    CONST robtarget rA_t278 := [[1931.75,1878.01,2213.21],[0.628788,0.0950822,0.552556,0.538765],[0,-2,-3,0],[9E+09,9E+09,9E+09,9E+09,9E+09,9E+09]];
    CONST robtarget rB_t278 := [[2895.21,136.965,1465.51],[0.672566,-0.676493,0.218304,-0.205806],[0,-3,2,0],[9E+09,9E+09,9E+09,9E+09,9E+09,9E+09]];
    CONST robtarget rB_t278_c1 := [[2895.21,136.965,1465.51],[0.672566,-0.676493,0.218304,-0.205806],[0,-4,-4,0],[9E+09,9E+09,9E+09,9E+09,9E+09,9E+09]];
    CONST robtarget rB_t278_c2 := [[2895.21,136.965,1465.51],[0.672566,-0.676493,0.218304,-0.205806],[0,0,-4,0],[9E+09,9E+09,9E+09,9E+09,9E+09,9E+09]];
    CONST jointtarget jA_t278 := [[44.9993,50.903,-73.3149,-90.0007,13.1401,-225.001],[9E+09,9E+09,9E+09,9E+09,9E+09,9E+09]];
    CONST jointtarget jB_t278 := [[0.000114317,56.0192,-54.9577,-270,55.0963,180],[9E+09,9E+09,9E+09,9E+09,9E+09,9E+09]];
    CONST jointtarget jBseed_t278 := [[0.000114414,56.0192,-54.9577,-270,55.0963,180],[9E+09,9E+09,9E+09,9E+09,9E+09,9E+09]];

    CONST robtarget rA_t279 := [[2895.21,136.965,1465.51],[0.672566,-0.676493,0.218304,-0.205806],[0,-3,2,0],[9E+09,9E+09,9E+09,9E+09,9E+09,9E+09]];
    CONST robtarget rB_t279 := [[1861.16,1900.88,2134.07],[0.550211,-0.0664014,0.550191,0.624619],[0,1,-2,0],[9E+09,9E+09,9E+09,9E+09,9E+09,9E+09]];
    CONST robtarget rB_t279_c4 := [[1861.16,1900.88,2134.07],[0.550211,-0.0664014,0.550191,0.624619],[0,-4,0,0],[9E+09,9E+09,9E+09,9E+09,9E+09,9E+09]];
    CONST robtarget rB_t279_c7 := [[1861.16,1900.88,2134.07],[0.550211,-0.0664014,0.550191,0.624619],[0,-4,4,0],[9E+09,9E+09,9E+09,9E+09,9E+09,9E+09]];
    CONST jointtarget jA_t279 := [[0.000114317,56.0192,-54.9577,-270,55.0963,180],[9E+09,9E+09,9E+09,9E+09,9E+09,9E+09]];
    CONST jointtarget jB_t279 := [[44.9999,40.5316,-53.7437,135,13.7626,-90.0002],[9E+09,9E+09,9E+09,9E+09,9E+09,9E+09]];
    CONST jointtarget jBseed_t279 := [[44.9999,40.5316,-53.7437,135,13.7626,-90.0001],[9E+09,9E+09,9E+09,9E+09,9E+09,9E+09]];

    CONST robtarget rA_t280 := [[1861.16,1900.88,2134.07],[0.550211,-0.0664014,0.550191,0.624619],[0,1,-2,0],[9E+09,9E+09,9E+09,9E+09,9E+09,9E+09]];
    CONST robtarget rB_t280 := [[89.7124,1202.36,2995.3],[0.131073,0.264977,0.137726,0.945325],[0,-2,2,0],[9E+09,9E+09,9E+09,9E+09,9E+09,9E+09]];
    CONST robtarget rB_t280_c1 := [[89.7124,1202.36,2995.3],[0.131073,0.264977,0.137726,0.945325],[0,-4,-4,0],[9E+09,9E+09,9E+09,9E+09,9E+09,9E+09]];
    CONST robtarget rB_t280_c2 := [[89.7124,1202.36,2995.3],[0.131073,0.264977,0.137726,0.945325],[0,0,-4,0],[9E+09,9E+09,9E+09,9E+09,9E+09,9E+09]];
    CONST jointtarget jA_t280 := [[44.9999,40.5316,-53.7437,135,13.7626,-90.0002],[9E+09,9E+09,9E+09,9E+09,9E+09,9E+09]];
    CONST jointtarget jB_t280 := [[89.999,-13.3177,-24.0516,-135.001,49.4253,224.999],[9E+09,9E+09,9E+09,9E+09,9E+09,9E+09]];
    CONST jointtarget jBseed_t280 := [[89.999,-13.3177,-24.0516,-135.001,49.4253,224.999],[9E+09,9E+09,9E+09,9E+09,9E+09,9E+09]];

    CONST robtarget rA_t281 := [[89.7124,1202.36,2995.3],[0.131073,0.264977,0.137726,0.945325],[0,-2,2,0],[9E+09,9E+09,9E+09,9E+09,9E+09,9E+09]];
    CONST robtarget rB_t281 := [[8.43678,485.853,3488.8],[0.00349083,0.0250045,0.137295,0.990208],[0,2,1,0],[9E+09,9E+09,9E+09,9E+09,9E+09,9E+09]];
    CONST robtarget rB_t281_c5 := [[8.43678,485.853,3488.8],[0.00349083,0.0250045,0.137295,0.990208],[0,0,0,0],[9E+09,9E+09,9E+09,9E+09,9E+09,9E+09]];
    CONST jointtarget jA_t281 := [[89.999,-13.3177,-24.0516,-135.001,49.4253,224.999],[9E+09,9E+09,9E+09,9E+09,9E+09,9E+09]];
    CONST jointtarget jB_t281 := [[89.9991,-5.53912,-68.673,269.999,2.89315,179.999],[9E+09,9E+09,9E+09,9E+09,9E+09,9E+09]];
    CONST jointtarget jBseed_t281 := [[89.9991,-5.53911,-68.6731,269.999,2.89315,179.999],[9E+09,9E+09,9E+09,9E+09,9E+09,9E+09]];

    CONST robtarget rA_t283 := [[-1405.69,-1439.34,2692.16],[0.0384433,0.29226,0.377677,-0.877762],[-2,1,2,0],[9E+09,9E+09,9E+09,9E+09,9E+09,9E+09]];
    CONST robtarget rB_t283 := [[812.974,-812.948,3221.93],[0.912154,0.146672,0.0607486,0.377853],[-1,2,-1,0],[9E+09,9E+09,9E+09,9E+09,9E+09,9E+09]];
    CONST robtarget rB_t283_c5 := [[812.974,-812.948,3221.93],[0.912154,0.146672,0.0607486,0.377853],[0,0,0,0],[9E+09,9E+09,9E+09,9E+09,9E+09,9E+09]];
    CONST robtarget rB_t283_c8 := [[812.974,-812.948,3221.93],[0.912154,0.146672,0.0607486,0.377853],[0,0,4,0],[9E+09,9E+09,9E+09,9E+09,9E+09,9E+09]];
    CONST jointtarget jA_t283 := [[-135,12.1897,-37.2472,135,11.6221,180],[9E+09,9E+09,9E+09,9E+09,9E+09,9E+09]];
    CONST jointtarget jB_t283 := [[-44.999,-5.94196,-41.7701,180.001,24.0187,-89.999],[9E+09,9E+09,9E+09,9E+09,9E+09,9E+09]];
    CONST jointtarget jBseed_t283 := [[-44.999,-5.94196,-41.7701,180.001,24.0187,-89.999],[9E+09,9E+09,9E+09,9E+09,9E+09,9E+09]];

    CONST robtarget rA_t284 := [[812.974,-812.948,3221.93],[0.912154,0.146672,0.0607486,0.377853],[-1,2,-1,0],[9E+09,9E+09,9E+09,9E+09,9E+09,9E+09]];
    CONST robtarget rB_t284 := [[1979.94,1852.8,2089.61],[0.764614,0.235393,0.316893,0.509445],[0,-2,-2,0],[9E+09,9E+09,9E+09,9E+09,9E+09,9E+09]];
    CONST robtarget rB_t284_c2 := [[1979.94,1852.8,2089.61],[0.764614,0.235393,0.316893,0.509445],[0,0,-4,0],[9E+09,9E+09,9E+09,9E+09,9E+09,9E+09]];
    CONST robtarget rB_t284_c3 := [[1979.94,1852.8,2089.61],[0.764614,0.235393,0.316893,0.509445],[0,4,-4,0],[9E+09,9E+09,9E+09,9E+09,9E+09,9E+09]];
    CONST jointtarget jA_t284 := [[-44.999,-5.94196,-41.7701,180.001,24.0187,-89.999],[9E+09,9E+09,9E+09,9E+09,9E+09,9E+09]];
    CONST jointtarget jB_t284 := [[45.0006,50.687,-65.7411,-134.999,49.5993,-179.999],[9E+09,9E+09,9E+09,9E+09,9E+09,9E+09]];
    CONST jointtarget jBseed_t284 := [[45.0006,50.687,-65.7411,-134.999,49.5993,-179.999],[9E+09,9E+09,9E+09,9E+09,9E+09,9E+09]];

    CONST robtarget rA_t286 := [[-1258.34,-1258.33,725.886],[0.308285,0.870927,-0.360749,-0.127697],[-2,-1,-4,0],[9E+09,9E+09,9E+09,9E+09,9E+09,9E+09]];
    CONST robtarget rB_t286 := [[767.091,-675.421,2450.3],[0.568653,0.350797,0.169976,0.72435],[-1,-3,-4,0],[9E+09,9E+09,9E+09,9E+09,9E+09,9E+09]];
    CONST robtarget rB_t286_c2 := [[767.091,-675.421,2450.3],[0.568653,0.350797,0.169976,0.72435],[0,0,-4,0],[9E+09,9E+09,9E+09,9E+09,9E+09,9E+09]];
    CONST jointtarget jA_t286 := [[-135,5.1912,38.7445,-0.000157696,7.07907,-270],[9E+09,9E+09,9E+09,9E+09,9E+09,9E+09]];
    CONST jointtarget jB_t286 := [[-44.9991,-40.7514,16.6024,-224.999,33.2841,-359.999],[9E+09,9E+09,9E+09,9E+09,9E+09,9E+09]];
    CONST jointtarget jBseed_t286 := [[-44.9991,-40.7514,16.6024,-224.999,33.2841,-359.999],[9E+09,9E+09,9E+09,9E+09,9E+09,9E+09]];

    CONST robtarget rA_t288 := [[-39.7659,1340.08,1419.52],[0.53573,-0.738869,-0.390158,-0.121829],[1,0,2,0],[9E+09,9E+09,9E+09,9E+09,9E+09,9E+09]];
    CONST robtarget rB_t288 := [[12.6582,1912.94,1121.44],[0.311805,-0.635779,-0.608576,-0.358048],[0,-1,2,0],[9E+09,9E+09,9E+09,9E+09,9E+09,9E+09]];
    CONST robtarget rB_t288_c5 := [[12.6582,1912.94,1121.44],[0.311805,-0.635779,-0.608576,-0.358048],[0,0,0,0],[9E+09,9E+09,9E+09,9E+09,9E+09,9E+09]];
    CONST jointtarget jA_t288 := [[90.0009,-37.8252,47.7227,45.0009,19.668,180.001],[9E+09,9E+09,9E+09,9E+09,9E+09,9E+09]];
    CONST jointtarget jB_t288 := [[89.9998,0.210577,28.8498,-45.0002,6.1507,225],[9E+09,9E+09,9E+09,9E+09,9E+09,9E+09]];
    CONST jointtarget jBseed_t288 := [[89.9998,0.210579,28.8498,-45.0002,6.1507,225],[9E+09,9E+09,9E+09,9E+09,9E+09,9E+09]];

    CONST robtarget rA_t290 := [[1406.56,-1559.53,2818.3],[0.150617,0.0701145,-0.509223,0.844447],[-1,3,-1,0],[9E+09,9E+09,9E+09,9E+09,9E+09,9E+09]];
    CONST robtarget rB_t290 := [[1821.8,-1916.48,1910.44],[0.145501,-0.116653,0.673226,-0.715534],[-1,2,-5,0],[9E+09,9E+09,9E+09,9E+09,9E+09,9E+09]];
    CONST robtarget rB_t290_c5 := [[1821.8,-1916.48,1910.44],[0.145501,-0.116653,0.673226,-0.715534],[0,0,0,0],[9E+09,9E+09,9E+09,9E+09,9E+09,9E+09]];
    CONST robtarget rB_t290_c6 := [[1821.8,-1916.48,1910.44],[0.145501,-0.116653,0.673226,-0.715534],[0,4,0,0],[9E+09,9E+09,9E+09,9E+09,9E+09,9E+09]];
    CONST jointtarget jA_t290 := [[-44.9996,31.5372,-69.78,270,40.376,-44.9996],[9E+09,9E+09,9E+09,9E+09,9E+09,9E+09]];
    CONST jointtarget jB_t290 := [[-45.0008,34.9614,-39.1119,269.999,23.6195,-360.001],[9E+09,9E+09,9E+09,9E+09,9E+09,9E+09]];
    CONST jointtarget jBseed_t290 := [[-45.0008,34.9614,-39.1119,269.999,23.6195,-360.001],[9E+09,9E+09,9E+09,9E+09,9E+09,9E+09]];

    CONST robtarget rA_t291 := [[1821.8,-1916.48,1910.44],[0.145501,-0.116653,0.673226,-0.715534],[-1,2,-5,0],[9E+09,9E+09,9E+09,9E+09,9E+09,9E+09]];
    CONST robtarget rB_t291 := [[50.5098,-2702.01,2116.99],[0.762943,0.487354,-0.0695059,0.419015],[-1,1,-4,0],[9E+09,9E+09,9E+09,9E+09,9E+09,9E+09]];
    CONST robtarget rB_t291_c5 := [[50.5098,-2702.01,2116.99],[0.762943,0.487354,-0.0695059,0.419015],[0,0,0,0],[9E+09,9E+09,9E+09,9E+09,9E+09,9E+09]];
    CONST jointtarget jA_t291 := [[-45.0008,34.9614,-39.1119,269.999,23.6195,-360.001],[9E+09,9E+09,9E+09,9E+09,9E+09,9E+09]];
    CONST jointtarget jB_t291 := [[-89.9996,45.3841,-59.6154,135,25.3151,-360],[9E+09,9E+09,9E+09,9E+09,9E+09,9E+09]];
    CONST jointtarget jBseed_t291 := [[-89.9996,45.3841,-59.6155,135,25.3151,-360],[9E+09,9E+09,9E+09,9E+09,9E+09,9E+09]];

    CONST robtarget rA_t293 := [[0.000160017,-2033.22,1759.97],[8.87382E-8,3.03818E-8,0.817508,-0.575917],[-1,0,3,0],[9E+09,9E+09,9E+09,9E+09,9E+09,9E+09]];
    CONST robtarget rB_t293 := [[-705.743,-705.745,3293.67],[2.528E-6,-0.101964,-0.101965,-0.989549],[-2,2,-3,0],[9E+09,9E+09,9E+09,9E+09,9E+09,9E+09]];
    CONST robtarget rB_t293_c5 := [[-705.743,-705.745,3293.67],[2.528E-6,-0.101964,-0.101965,-0.989549],[0,0,0,0],[9E+09,9E+09,9E+09,9E+09,9E+09,9E+09]];
    CONST jointtarget jA_t293 := [[-90,-0.214244,6.61641,9.73535E-6,13.2701,270],[9E+09,9E+09,9E+09,9E+09,9E+09,9E+09]];
    CONST jointtarget jB_t293 := [[-135,-3.3015,-48.9074,180,54.373,-225],[9E+09,9E+09,9E+09,9E+09,9E+09,9E+09]];
    CONST jointtarget jBseed_t293 := [[-135,-3.30149,-48.9074,180,54.373,-225],[9E+09,9E+09,9E+09,9E+09,9E+09,9E+09]];

    CONST robtarget rA_t294 := [[-705.743,-705.745,3293.67],[2.528E-6,-0.101964,-0.101965,-0.989549],[-2,2,-3,0],[9E+09,9E+09,9E+09,9E+09,9E+09,9E+09]];
    CONST robtarget rB_t294 := [[-1094.14,-971.928,9.47825],[0.208069,-0.895798,-0.340492,0.195752],[-2,3,1,0],[9E+09,9E+09,9E+09,9E+09,9E+09,9E+09]];
    CONST robtarget rB_t294_c3 := [[-1094.14,-971.928,9.47825],[0.208069,-0.895798,-0.340492,0.195752],[0,4,-4,0],[9E+09,9E+09,9E+09,9E+09,9E+09,9E+09]];
    CONST jointtarget jA_t294 := [[-135,-3.3015,-48.9074,180,54.373,-225],[9E+09,9E+09,9E+09,9E+09,9E+09,9E+09]];
    CONST jointtarget jB_t294 := [[-135,31.9108,46.0247,270,31.1655,90.0004],[9E+09,9E+09,9E+09,9E+09,9E+09,9E+09]];
    CONST jointtarget jBseed_t294 := [[-135,31.9108,46.0247,270,31.1655,90.0004],[9E+09,9E+09,9E+09,9E+09,9E+09,9E+09]];

    CONST robtarget rA_t295 := [[-1094.14,-971.928,9.47825],[0.208069,-0.895798,-0.340492,0.195752],[-2,3,1,0],[9E+09,9E+09,9E+09,9E+09,9E+09,9E+09]];
    CONST robtarget rB_t295 := [[-0.0128204,-2555.07,2364.03],[0.379873,0.046241,0.111641,-0.917112],[-2,-3,1,0],[9E+09,9E+09,9E+09,9E+09,9E+09,9E+09]];
    CONST robtarget rB_t295_c5 := [[-0.0128204,-2555.07,2364.03],[0.379873,0.046241,0.111641,-0.917112],[0,0,0,0],[9E+09,9E+09,9E+09,9E+09,9E+09,9E+09]];
    CONST jointtarget jA_t295 := [[-135,31.9108,46.0247,270,31.1655,90.0004],[9E+09,9E+09,9E+09,9E+09,9E+09,9E+09]];
    CONST jointtarget jB_t295 := [[-90.0003,51.5513,-76.5603,-180,51.1099,135],[9E+09,9E+09,9E+09,9E+09,9E+09,9E+09]];
    CONST jointtarget jBseed_t295 := [[-90.0003,51.5513,-76.5603,-180,51.11,135],[9E+09,9E+09,9E+09,9E+09,9E+09,9E+09]];

    CONST robtarget rA_t296 := [[-0.0128204,-2555.07,2364.03],[0.379873,0.046241,0.111641,-0.917112],[-2,-3,1,0],[9E+09,9E+09,9E+09,9E+09,9E+09,9E+09]];
    CONST robtarget rB_t296 := [[-133.882,-1999.9,2604.31],[0.245559,-0.3752,-0.489462,0.747899],[-2,-2,-1,0],[9E+09,9E+09,9E+09,9E+09,9E+09,9E+09]];
    CONST robtarget rB_t296_c5 := [[-133.882,-1999.9,2604.31],[0.245559,-0.3752,-0.489462,0.747899],[0,0,0,0],[9E+09,9E+09,9E+09,9E+09,9E+09,9E+09]];
    CONST jointtarget jA_t296 := [[-90.0003,51.5513,-76.5603,-180,51.1099,135],[9E+09,9E+09,9E+09,9E+09,9E+09,9E+09]];
    CONST jointtarget jB_t296 := [[-90.0004,12.9148,-36.5093,-90.0004,53.2835,-0.000410538],[9E+09,9E+09,9E+09,9E+09,9E+09,9E+09]];
    CONST jointtarget jBseed_t296 := [[-90.0004,12.9148,-36.5093,-90.0004,53.2835,-0.000407697],[9E+09,9E+09,9E+09,9E+09,9E+09,9E+09]];

    CONST robtarget rA_t297 := [[-133.882,-1999.9,2604.31],[0.245559,-0.3752,-0.489462,0.747899],[-2,-2,-1,0],[9E+09,9E+09,9E+09,9E+09,9E+09,9E+09]];
    CONST robtarget rB_t297 := [[1996.66,-62.2443,1865.38],[0.57107,0.599825,0.416979,0.374455],[0,3,-2,0],[9E+09,9E+09,9E+09,9E+09,9E+09,9E+09]];
    CONST robtarget rB_t297_c2 := [[1996.66,-62.2443,1865.38],[0.57107,0.599825,0.416979,0.374455],[0,0,-4,0],[9E+09,9E+09,9E+09,9E+09,9E+09,9E+09]];
    CONST robtarget rB_t297_c5 := [[1996.66,-62.2443,1865.38],[0.57107,0.599825,0.416979,0.374455],[0,0,0,0],[9E+09,9E+09,9E+09,9E+09,9E+09,9E+09]];
    CONST jointtarget jA_t297 := [[-90.0004,12.9148,-36.5093,-90.0004,53.2835,-0.000410538],[9E+09,9E+09,9E+09,9E+09,9E+09,9E+09]];
    CONST jointtarget jB_t297 := [[0.000436422,-1.83294,5.99353,270,21.8891,-180],[9E+09,9E+09,9E+09,9E+09,9E+09,9E+09]];
    CONST jointtarget jBseed_t297 := [[0.000436628,-1.83294,5.99353,270,21.8891,-180],[9E+09,9E+09,9E+09,9E+09,9E+09,9E+09]];

    CONST robtarget rA_t298 := [[1996.66,-62.2443,1865.38],[0.57107,0.599825,0.416979,0.374455],[0,3,-2,0],[9E+09,9E+09,9E+09,9E+09,9E+09,9E+09]];
    CONST robtarget rB_t298 := [[-0.0358595,2407.99,2512.57],[0.694216,-0.134324,0.134333,0.694245],[1,2,2,0],[9E+09,9E+09,9E+09,9E+09,9E+09,9E+09]];
    CONST robtarget rB_t298_c2 := [[-0.0358595,2407.99,2512.57],[0.694216,-0.134324,0.134333,0.694245],[0,0,-4,0],[9E+09,9E+09,9E+09,9E+09,9E+09,9E+09]];
    CONST jointtarget jA_t298 := [[0.000436422,-1.83294,5.99353,270,21.8891,-180],[9E+09,9E+09,9E+09,9E+09,9E+09,9E+09]];
    CONST jointtarget jB_t298 := [[90.0009,37.9388,-61.6031,180.001,44.4337,180.001],[9E+09,9E+09,9E+09,9E+09,9E+09,9E+09]];
    CONST jointtarget jBseed_t298 := [[90.0009,37.9388,-61.6031,180.001,44.4337,180.001],[9E+09,9E+09,9E+09,9E+09,9E+09,9E+09]];

    CONST robtarget rA_t299 := [[-0.0358595,2407.99,2512.57],[0.694216,-0.134324,0.134333,0.694245],[1,2,2,0],[9E+09,9E+09,9E+09,9E+09,9E+09,9E+09]];
    CONST robtarget rB_t299 := [[0.0269352,2024.98,2914.37],[0.65455,-0.267481,-0.267485,-0.654576],[0,-3,3,0],[9E+09,9E+09,9E+09,9E+09,9E+09,9E+09]];
    CONST robtarget rB_t299_c5 := [[0.0269352,2024.98,2914.37],[0.65455,-0.267481,-0.267485,-0.654576],[0,0,0,0],[9E+09,9E+09,9E+09,9E+09,9E+09,9E+09]];
    CONST robtarget rB_t299_c8 := [[0.0269352,2024.98,2914.37],[0.65455,-0.267481,-0.267485,-0.654576],[0,0,4,0],[9E+09,9E+09,9E+09,9E+09,9E+09,9E+09]];
    CONST jointtarget jA_t299 := [[90.0009,37.9388,-61.6031,180.001,44.4337,180.001],[9E+09,9E+09,9E+09,9E+09,9E+09,9E+09]];
    CONST jointtarget jB_t299 := [[89.9992,27.0766,-66.003,-180.001,6.61947,359.999],[9E+09,9E+09,9E+09,9E+09,9E+09,9E+09]];
    CONST jointtarget jBseed_t299 := [[89.9992,27.0766,-66.003,-180.001,6.61946,359.999],[9E+09,9E+09,9E+09,9E+09,9E+09,9E+09]];

    CONST robtarget rA_t301 := [[711.687,820.474,2264.17],[0.740004,-0.357438,-0.197934,-0.534279],[0,1,-4,0],[9E+09,9E+09,9E+09,9E+09,9E+09,9E+09]];
    CONST robtarget rB_t301 := [[-794.783,716.383,3401.08],[0.401784,0.232779,-0.132142,-0.875741],[1,-4,-1,0],[9E+09,9E+09,9E+09,9E+09,9E+09,9E+09]];
    CONST robtarget rB_t301_c5 := [[-794.783,716.383,3401.08],[0.401784,0.232779,-0.132142,-0.875741],[0,0,0,0],[9E+09,9E+09,9E+09,9E+09,9E+09,9E+09]];
    CONST jointtarget jA_t301 := [[44.9993,-42.165,24.799,134.999,40.6561,-270.001],[9E+09,9E+09,9E+09,9E+09,9E+09,9E+09]];
    CONST jointtarget jB_t301 := [[135,11.1533,-76.4135,-270,19.3896,-0.000262528],[9E+09,9E+09,9E+09,9E+09,9E+09,9E+09]];
    CONST jointtarget jBseed_t301 := [[135,11.1533,-76.4135,-270,19.3896,-0.000243019],[9E+09,9E+09,9E+09,9E+09,9E+09,9E+09]];

    CONST robtarget rA_t303 := [[-1207.94,-1217.23,2595.23],[0.584806,0.577737,0.0162937,-0.569172],[-2,0,3,0],[9E+09,9E+09,9E+09,9E+09,9E+09,9E+09]];
    CONST robtarget rB_t303 := [[-1933.3,-2020.07,1434.77],[0.640752,0.612752,-0.440334,0.141698],[-2,-3,0,0],[9E+09,9E+09,9E+09,9E+09,9E+09,9E+09]];
    CONST robtarget rB_t303_c5 := [[-1933.3,-2020.07,1434.77],[0.640752,0.612752,-0.440334,0.141698],[0,0,0,0],[9E+09,9E+09,9E+09,9E+09,9E+09,9E+09]];
    CONST jointtarget jA_t303 := [[-135,-6.5096,-15.1488,44.9998,3.19163,360],[9E+09,9E+09,9E+09,9E+09,9E+09,9E+09]];
    CONST jointtarget jB_t303 := [[-135,42.8608,-34.2836,-270,21.5467,45.0005],[9E+09,9E+09,9E+09,9E+09,9E+09,9E+09]];
    CONST jointtarget jBseed_t303 := [[-135,42.8608,-34.2836,-270,21.5467,45.0005],[9E+09,9E+09,9E+09,9E+09,9E+09,9E+09]];

    CONST robtarget rA_t306 := [[-0.00435252,-1330.24,-413.892],[0.081587,0.373884,0.902639,-0.196969],[-2,1,-3,0],[9E+09,9E+09,9E+09,9E+09,9E+09,9E+09]];
    CONST robtarget rB_t306 := [[1109.78,-1031.5,1346.08],[0.314617,0.796486,0.0990844,0.506762],[-1,0,0,0],[9E+09,9E+09,9E+09,9E+09,9E+09,9E+09]];
    CONST robtarget rB_t306_c2 := [[1109.78,-1031.5,1346.08],[0.314617,0.796486,0.0990844,0.506762],[0,0,-4,0],[9E+09,9E+09,9E+09,9E+09,9E+09,9E+09]];
    CONST robtarget rB_t306_c5 := [[1109.78,-1031.5,1346.08],[0.314617,0.796486,0.0990844,0.506762],[0,0,0,0],[9E+09,9E+09,9E+09,9E+09,9E+09,9E+09]];
    CONST jointtarget jA_t306 := [[-90.0002,55.88,40.99,180,31.4896,-225],[9E+09,9E+09,9E+09,9E+09,9E+09,9E+09]];
    CONST jointtarget jB_t306 := [[-45.0005,-25.9706,43.7712,89.9995,19.3622,44.9995],[9E+09,9E+09,9E+09,9E+09,9E+09,9E+09]];
    CONST jointtarget jBseed_t306 := [[-45.0005,-25.9706,43.7712,89.9995,19.3622,44.9995],[9E+09,9E+09,9E+09,9E+09,9E+09,9E+09]];

    CONST robtarget rA_t307 := [[1109.78,-1031.5,1346.08],[0.314617,0.796486,0.0990844,0.506762],[-1,0,0,0],[9E+09,9E+09,9E+09,9E+09,9E+09,9E+09]];
    CONST robtarget rB_t307 := [[1813.28,-1813.32,1534.44],[0.580903,0.575562,0.575569,-1.19777E-5],[-1,-1,0,0],[9E+09,9E+09,9E+09,9E+09,9E+09,9E+09]];
    CONST robtarget rB_t307_c5 := [[1813.28,-1813.32,1534.44],[0.580903,0.575562,0.575569,-1.19777E-5],[0,0,0,0],[9E+09,9E+09,9E+09,9E+09,9E+09,9E+09]];
    CONST jointtarget jA_t307 := [[-45.0005,-25.9706,43.7712,89.9995,19.3622,44.9995],[9E+09,9E+09,9E+09,9E+09,9E+09,9E+09]];
    CONST jointtarget jB_t307 := [[-45.0007,28.1057,-18.1997,-0.000729667,9.06583,44.9993],[9E+09,9E+09,9E+09,9E+09,9E+09,9E+09]];
    CONST jointtarget jBseed_t307 := [[-45.0007,28.1057,-18.1997,-0.000737297,9.06583,44.9993],[9E+09,9E+09,9E+09,9E+09,9E+09,9E+09]];

    CONST robtarget rA_t308 := [[1813.28,-1813.32,1534.44],[0.580903,0.575562,0.575569,-1.19777E-5],[-1,-1,0,0],[9E+09,9E+09,9E+09,9E+09,9E+09,9E+09]];
    CONST robtarget rB_t308 := [[2140.65,93.5238,2492.89],[0.519043,-0.360662,-0.121204,-0.765393],[0,-3,-3,0],[9E+09,9E+09,9E+09,9E+09,9E+09,9E+09]];
    CONST robtarget rB_t308_c4 := [[2140.65,93.5238,2492.89],[0.519043,-0.360662,-0.121204,-0.765393],[0,-4,0,0],[9E+09,9E+09,9E+09,9E+09,9E+09,9E+09]];
    CONST robtarget rB_t308_c5 := [[2140.65,93.5238,2492.89],[0.519043,-0.360662,-0.121204,-0.765393],[0,0,0,0],[9E+09,9E+09,9E+09,9E+09,9E+09,9E+09]];
    CONST jointtarget jA_t308 := [[-45.0007,28.1057,-18.1997,-0.000729667,9.06583,44.9993],[9E+09,9E+09,9E+09,9E+09,9E+09,9E+09]];
    CONST jointtarget jB_t308 := [[0.000401838,16.7455,-33.264,-225,52.3606,-270],[9E+09,9E+09,9E+09,9E+09,9E+09,9E+09]];
    CONST jointtarget jBseed_t308 := [[0.000401837,16.7455,-33.264,-225,52.3606,-270],[9E+09,9E+09,9E+09,9E+09,9E+09,9E+09]];

    CONST robtarget rA_t311 := [[-1668.51,-1668.47,341.824],[0.590053,0.294475,-0.710909,0.2444],[-2,-3,3,0],[9E+09,9E+09,9E+09,9E+09,9E+09,9E+09]];
    CONST robtarget rB_t311 := [[1659.54,-1659.53,736.873],[0.559459,7.7831E-7,0.611567,-0.559457],[-1,-2,-3,0],[9E+09,9E+09,9E+09,9E+09,9E+09,9E+09]];
    CONST robtarget rB_t311_c4 := [[1659.54,-1659.53,736.873],[0.559459,7.7831E-7,0.611567,-0.559457],[0,-4,0,0],[9E+09,9E+09,9E+09,9E+09,9E+09,9E+09]];
    CONST jointtarget jA_t311 := [[-135.001,43.7764,8.73104,-180.001,41.8922,359.999],[9E+09,9E+09,9E+09,9E+09,9E+09,9E+09]];
    CONST jointtarget jB_t311 := [[-44.9999,32.6286,10.7941,-180,58.0169,-225],[9E+09,9E+09,9E+09,9E+09,9E+09,9E+09]];
    CONST jointtarget jBseed_t311 := [[-44.9999,32.6286,10.7941,-180,58.0169,-225],[9E+09,9E+09,9E+09,9E+09,9E+09,9E+09]];

    CONST robtarget rA_t316 := [[31.8866,-661.423,2881.06],[0.650157,0.260758,0.387274,-0.599433],[-2,0,-1,0],[9E+09,9E+09,9E+09,9E+09,9E+09,9E+09]];
    CONST robtarget rB_t316 := [[67.0004,-1549.03,-423.181],[0.0272108,0.674661,0.686619,0.269531],[-1,0,-1,0],[9E+09,9E+09,9E+09,9E+09,9E+09,9E+09]];
    CONST robtarget rB_t316_c5 := [[67.0004,-1549.03,-423.181],[0.0272108,0.674661,0.686619,0.269531],[0,0,0,0],[9E+09,9E+09,9E+09,9E+09,9E+09,9E+09]];
    CONST jointtarget jA_t316 := [[-90.0005,-39.8358,-6.45618,44.9995,15.6688,-45.0005],[9E+09,9E+09,9E+09,9E+09,9E+09,9E+09]];
    CONST jointtarget jB_t316 := [[-89.9991,59.0698,26.3106,45.0009,34.5531,-44.9991],[9E+09,9E+09,9E+09,9E+09,9E+09,9E+09]];
    CONST jointtarget jBseed_t316 := [[-89.9991,59.0698,26.3106,45.0009,34.5531,-44.9991],[9E+09,9E+09,9E+09,9E+09,9E+09,9E+09]];

    CONST robtarget rA_t317 := [[67.0004,-1549.03,-423.181],[0.0272108,0.674661,0.686619,0.269531],[-1,0,-1,0],[9E+09,9E+09,9E+09,9E+09,9E+09,9E+09]];
    CONST robtarget rB_t317 := [[1093.81,-961.271,-433.788],[0.203083,0.00193774,0.955933,0.212005],[-1,-3,-2,0],[9E+09,9E+09,9E+09,9E+09,9E+09,9E+09]];
    CONST robtarget rB_t317_c5 := [[1093.81,-961.271,-433.788],[0.203083,0.00193774,0.955933,0.212005],[0,0,0,0],[9E+09,9E+09,9E+09,9E+09,9E+09,9E+09]];
    CONST robtarget rB_t317_c8 := [[1093.81,-961.271,-433.788],[0.203083,0.00193774,0.955933,0.212005],[0,0,4,0],[9E+09,9E+09,9E+09,9E+09,9E+09,9E+09]];
    CONST jointtarget jA_t317 := [[-89.9991,59.0698,26.3106,45.0009,34.5531,-44.9991],[9E+09,9E+09,9E+09,9E+09,9E+09,9E+09]];
    CONST jointtarget jB_t317 := [[-44.9999,58.5461,32.2102,-270,34.1374,-135],[9E+09,9E+09,9E+09,9E+09,9E+09,9E+09]];
    CONST jointtarget jBseed_t317 := [[-44.9999,58.5461,32.2102,-270,34.1374,-135],[9E+09,9E+09,9E+09,9E+09,9E+09,9E+09]];

    CONST robtarget rA_t319 := [[-247.85,152.002,3494.48],[0.3863,0.144348,0.205674,-0.887488],[1,-3,-1,0],[9E+09,9E+09,9E+09,9E+09,9E+09,9E+09]];
    CONST robtarget rB_t319 := [[1522.3,1582.86,1574.78],[0.437235,-0.846027,-0.0820903,-0.293813],[0,0,1,0],[9E+09,9E+09,9E+09,9E+09,9E+09,9E+09]];
    CONST robtarget rB_t319_c2 := [[1522.3,1582.86,1574.78],[0.437235,-0.846027,-0.0820903,-0.293813],[0,0,-4,0],[9E+09,9E+09,9E+09,9E+09,9E+09,9E+09]];
    CONST jointtarget jA_t319 := [[135.001,-2.30911,-78.3931,-224.999,35.0237,-44.9992],[9E+09,9E+09,9E+09,9E+09,9E+09,9E+09]];
    CONST jointtarget jB_t319 := [[44.9998,9.10246,2.92276,44.9998,21.2665,180],[9E+09,9E+09,9E+09,9E+09,9E+09,9E+09]];
    CONST jointtarget jBseed_t319 := [[44.9998,9.10246,2.92276,44.9998,21.2665,180],[9E+09,9E+09,9E+09,9E+09,9E+09,9E+09]];

    CONST robtarget rA_t320 := [[1522.3,1582.86,1574.78],[0.437235,-0.846027,-0.0820903,-0.293813],[0,0,1,0],[9E+09,9E+09,9E+09,9E+09,9E+09,9E+09]];
    CONST robtarget rB_t320 := [[29.1179,-2091.95,2261.12],[0.459763,0.544345,-0.448947,0.539215],[-1,0,1,0],[9E+09,9E+09,9E+09,9E+09,9E+09,9E+09]];
    CONST robtarget rB_t320_c5 := [[29.1179,-2091.95,2261.12],[0.459763,0.544345,-0.448947,0.539215],[0,0,0,0],[9E+09,9E+09,9E+09,9E+09,9E+09,9E+09]];
    CONST jointtarget jA_t320 := [[44.9998,9.10246,2.92276,44.9998,21.2665,180],[9E+09,9E+09,9E+09,9E+09,9E+09,9E+09]];
    CONST jointtarget jB_t320 := [[-89.9993,6.24591,-16.6842,45.0007,14.2625,135.001],[9E+09,9E+09,9E+09,9E+09,9E+09,9E+09]];
    CONST jointtarget jBseed_t320 := [[-89.9993,6.24592,-16.6842,45.0007,14.2625,135.001],[9E+09,9E+09,9E+09,9E+09,9E+09,9E+09]];

    CONST robtarget rA_t322 := [[-0.0284785,1965.77,2672.38],[1.9163E-5,-6.84607E-6,-0.149469,-0.988766],[1,2,3,0],[9E+09,9E+09,9E+09,9E+09,9E+09,9E+09]];
    CONST robtarget rB_t322 := [[42.8658,1982.85,2907.31],[0.887318,-0.257326,0.232757,0.303767],[1,-2,-3,0],[9E+09,9E+09,9E+09,9E+09,9E+09,9E+09]];
    CONST robtarget rB_t322_c6 := [[42.8658,1982.85,2907.31],[0.887318,-0.257326,0.232757,0.303767],[0,4,0,0],[9E+09,9E+09,9E+09,9E+09,9E+09,9E+09]];
    CONST jointtarget jA_t322 := [[90.0009,11.6331,-32.8236,180.001,51.6172,270.001],[9E+09,9E+09,9E+09,9E+09,9E+09,9E+09]];
    CONST jointtarget jB_t322 := [[90.0002,22.8797,-59.2465,-135,21.2885,-270],[9E+09,9E+09,9E+09,9E+09,9E+09,9E+09]];
    CONST jointtarget jBseed_t322 := [[90.0002,22.8797,-59.2465,-135,21.2885,-270],[9E+09,9E+09,9E+09,9E+09,9E+09,9E+09]];

    CONST robtarget rA_t323 := [[42.8658,1982.85,2907.31],[0.887318,-0.257326,0.232757,0.303767],[1,-2,-3,0],[9E+09,9E+09,9E+09,9E+09,9E+09,9E+09]];
    CONST robtarget rB_t323 := [[1926.37,1926.36,1610.82],[0.743075,-0.473202,0.473201,-1.62968E-6],[0,-3,1,0],[9E+09,9E+09,9E+09,9E+09,9E+09,9E+09]];
    CONST robtarget rB_t323_c1 := [[1926.37,1926.36,1610.82],[0.743075,-0.473202,0.473201,-1.62968E-6],[0,-4,-4,0],[9E+09,9E+09,9E+09,9E+09,9E+09,9E+09]];
    CONST jointtarget jA_t323 := [[90.0002,22.8797,-59.2465,-135,21.2885,-270],[9E+09,9E+09,9E+09,9E+09,9E+09,9E+09]];
    CONST jointtarget jB_t323 := [[44.9999,37.2649,-31.0779,-180,12.1751,135],[9E+09,9E+09,9E+09,9E+09,9E+09,9E+09]];
    CONST jointtarget jBseed_t323 := [[44.9999,37.2649,-31.0779,-180,12.1751,135],[9E+09,9E+09,9E+09,9E+09,9E+09,9E+09]];

    CONST robtarget rA_t325 := [[993.69,1029.26,2606.44],[0.592567,-0.598865,-0.0638388,-0.534929],[0,0,1,0],[9E+09,9E+09,9E+09,9E+09,9E+09,9E+09]];
    CONST robtarget rB_t325 := [[2370.61,92.2602,2505.16],[0.805262,-0.421768,0.382388,-0.165663],[-1,0,2,0],[9E+09,9E+09,9E+09,9E+09,9E+09,9E+09]];
    CONST robtarget rB_t325_c2 := [[2370.61,92.2602,2505.16],[0.805262,-0.421768,0.382388,-0.165663],[0,0,-4,0],[9E+09,9E+09,9E+09,9E+09,9E+09,9E+09]];
    CONST robtarget rB_t325_c5 := [[2370.61,92.2602,2505.16],[0.805262,-0.421768,0.382388,-0.165663],[0,0,0,0],[9E+09,9E+09,9E+09,9E+09,9E+09,9E+09]];
    CONST jointtarget jA_t325 := [[44.9999,-19.1699,-5.71824,45,12.2977,180],[9E+09,9E+09,9E+09,9E+09,9E+09,9E+09]];
    CONST jointtarget jB_t325 := [[-0.000494033,32.7531,-57.7191,89.9995,33.5441,225],[9E+09,9E+09,9E+09,9E+09,9E+09,9E+09]];
    CONST jointtarget jBseed_t325 := [[-0.000494125,32.7531,-57.719,89.9995,33.5441,225],[9E+09,9E+09,9E+09,9E+09,9E+09,9E+09]];

    CONST robtarget rA_t326 := [[2370.61,92.2602,2505.16],[0.805262,-0.421768,0.382388,-0.165663],[-1,0,2,0],[9E+09,9E+09,9E+09,9E+09,9E+09,9E+09]];
    CONST robtarget rB_t326 := [[-74.1318,1962.29,1808.92],[0.43485,-0.505503,0.288513,0.687119],[1,-3,2,0],[9E+09,9E+09,9E+09,9E+09,9E+09,9E+09]];
    CONST robtarget rB_t326_c5 := [[-74.1318,1962.29,1808.92],[0.43485,-0.505503,0.288513,0.687119],[0,0,0,0],[9E+09,9E+09,9E+09,9E+09,9E+09,9E+09]];
    CONST robtarget rB_t326_c8 := [[-74.1318,1962.29,1808.92],[0.43485,-0.505503,0.288513,0.687119],[0,0,4,0],[9E+09,9E+09,9E+09,9E+09,9E+09,9E+09]];
    CONST jointtarget jA_t326 := [[-0.000494033,32.7531,-57.7191,89.9995,33.5441,225],[9E+09,9E+09,9E+09,9E+09,9E+09,9E+09]];
    CONST jointtarget jB_t326 := [[90.0007,-2.93527,11.5281,-224.999,38.8708,225.001],[9E+09,9E+09,9E+09,9E+09,9E+09,9E+09]];
    CONST jointtarget jBseed_t326 := [[90.0007,-2.93527,11.5281,-224.999,38.8708,225.001],[9E+09,9E+09,9E+09,9E+09,9E+09,9E+09]];

    CONST robtarget rA_t327 := [[-74.1318,1962.29,1808.92],[0.43485,-0.505503,0.288513,0.687119],[1,-3,2,0],[9E+09,9E+09,9E+09,9E+09,9E+09,9E+09]];
    CONST robtarget rB_t327 := [[541.561,58.9595,3221.16],[0.594968,0.173633,0.423525,0.660675],[0,0,-4,0],[9E+09,9E+09,9E+09,9E+09,9E+09,9E+09]];
    CONST robtarget rB_t327_c5 := [[541.561,58.9595,3221.16],[0.594968,0.173633,0.423525,0.660675],[0,0,0,0],[9E+09,9E+09,9E+09,9E+09,9E+09,9E+09]];
    CONST jointtarget jA_t327 := [[90.0007,-2.93527,11.5281,-224.999,38.8708,225.001],[9E+09,9E+09,9E+09,9E+09,9E+09,9E+09]];
    CONST jointtarget jB_t327 := [[0.000888097,-25.8095,-34.7398,45.0009,29.9478,-314.999],[9E+09,9E+09,9E+09,9E+09,9E+09,9E+09]];
    CONST jointtarget jBseed_t327 := [[0.000887081,-25.8095,-34.7398,45.0009,29.9478,-314.999],[9E+09,9E+09,9E+09,9E+09,9E+09,9E+09]];

    CONST robtarget rA_t328 := [[541.561,58.9595,3221.16],[0.594968,0.173633,0.423525,0.660675],[0,0,-4,0],[9E+09,9E+09,9E+09,9E+09,9E+09,9E+09]];
    CONST robtarget rB_t328 := [[1048.64,-0.0107856,1817.23],[0.331673,-0.460805,0.190867,-0.800763],[-1,-3,0,0],[9E+09,9E+09,9E+09,9E+09,9E+09,9E+09]];
    CONST robtarget rB_t328_c2 := [[1048.64,-0.0107856,1817.23],[0.331673,-0.460805,0.190867,-0.800763],[0,0,-4,0],[9E+09,9E+09,9E+09,9E+09,9E+09,9E+09]];
    CONST jointtarget jA_t328 := [[0.000888097,-25.8095,-34.7398,45.0009,29.9478,-314.999],[9E+09,9E+09,9E+09,9E+09,9E+09,9E+09]];
    CONST jointtarget jB_t328 := [[-0.000625985,-55.0523,46.7348,-180.001,21.8451,44.9994],[9E+09,9E+09,9E+09,9E+09,9E+09,9E+09]];
    CONST jointtarget jBseed_t328 := [[-0.000626026,-55.0523,46.7348,-180.001,21.8451,44.9994],[9E+09,9E+09,9E+09,9E+09,9E+09,9E+09]];

    CONST robtarget rA_t330 := [[1979.03,1927.94,2111.66],[0.535364,-0.563616,0.0896725,-0.622641],[0,-1,-1,0],[9E+09,9E+09,9E+09,9E+09,9E+09,9E+09]];
    CONST robtarget rB_t330 := [[0.0266284,-1625.03,2883.01],[0.729771,0.566569,0.234678,-0.302259],[-1,0,0,0],[9E+09,9E+09,9E+09,9E+09,9E+09,9E+09]];
    CONST robtarget rB_t330_c2 := [[0.0266284,-1625.03,2883.01],[0.729771,0.566569,0.234678,-0.302259],[0,0,-4,0],[9E+09,9E+09,9E+09,9E+09,9E+09,9E+09]];
    CONST robtarget rB_t330_c5 := [[0.0266284,-1625.03,2883.01],[0.729771,0.566569,0.234678,-0.302259],[0,0,0,0],[9E+09,9E+09,9E+09,9E+09,9E+09,9E+09]];
    CONST jointtarget jA_t330 := [[45.0004,54.8949,-75.8144,-89.9996,12.4992,-44.9997],[9E+09,9E+09,9E+09,9E+09,9E+09,9E+09]];
    CONST jointtarget jB_t330 := [[-89.9991,-0.485245,-34.5256,0.000901937,20.6604,45.0009],[9E+09,9E+09,9E+09,9E+09,9E+09,9E+09]];
    CONST jointtarget jBseed_t330 := [[-89.9991,-0.485245,-34.5256,0.000909116,20.6604,45.0009],[9E+09,9E+09,9E+09,9E+09,9E+09,9E+09]];

    CONST robtarget rA_t331 := [[0.0266284,-1625.03,2883.01],[0.729771,0.566569,0.234678,-0.302259],[-1,0,0,0],[9E+09,9E+09,9E+09,9E+09,9E+09,9E+09]];
    CONST robtarget rB_t331 := [[9.32158,-1659.97,1095.82],[0.170899,0.343219,-0.791669,0.475661],[-2,0,1,0],[9E+09,9E+09,9E+09,9E+09,9E+09,9E+09]];
    CONST robtarget rB_t331_c2 := [[9.32158,-1659.97,1095.82],[0.170899,0.343219,-0.791669,0.475661],[0,0,-4,0],[9E+09,9E+09,9E+09,9E+09,9E+09,9E+09]];
    CONST robtarget rB_t331_c5 := [[9.32158,-1659.97,1095.82],[0.170899,0.343219,-0.791669,0.475661],[0,0,0,0],[9E+09,9E+09,9E+09,9E+09,9E+09,9E+09]];
    CONST jointtarget jA_t331 := [[-89.9991,-0.485245,-34.5256,0.000901937,20.6604,45.0009],[9E+09,9E+09,9E+09,9E+09,9E+09,9E+09]];
    CONST jointtarget jB_t331 := [[-90.0006,-13.0284,42.3588,89.9993,3.20627,134.999],[9E+09,9E+09,9E+09,9E+09,9E+09,9E+09]];
    CONST jointtarget jBseed_t331 := [[-90.0006,-13.0284,42.3588,89.9994,3.20627,134.999],[9E+09,9E+09,9E+09,9E+09,9E+09,9E+09]];

    CONST robtarget rA_t336 := [[-1130.21,1052.11,2680.84],[0.872347,-0.016871,-0.413391,-0.260448],[1,1,0,0],[9E+09,9E+09,9E+09,9E+09,9E+09,9E+09]];
    CONST robtarget rB_t336 := [[1324.12,1324.12,2692.34],[2.37779E-6,0.141217,0.141218,0.979855],[0,-3,-1,0],[9E+09,9E+09,9E+09,9E+09,9E+09,9E+09]];
    CONST robtarget rB_t336_c5 := [[1324.12,1324.12,2692.34],[2.37779E-6,0.141217,0.141218,0.979855],[0,0,0,0],[9E+09,9E+09,9E+09,9E+09,9E+09,9E+09]];
    CONST robtarget rB_t336_c8 := [[1324.12,1324.12,2692.34],[2.37779E-6,0.141217,0.141218,0.979855],[0,0,4,0],[9E+09,9E+09,9E+09,9E+09,9E+09,9E+09]];
    CONST jointtarget jA_t336 := [[135,-11.6953,-11.9669,135,27.8842,44.9999],[9E+09,9E+09,9E+09,9E+09,9E+09,9E+09]];
    CONST jointtarget jB_t336 := [[44.9999,6.24592,-27.8326,-180,45.3731,-45.0001],[9E+09,9E+09,9E+09,9E+09,9E+09,9E+09]];
    CONST jointtarget jBseed_t336 := [[44.9999,6.24592,-27.8326,-180,45.3731,-45.0001],[9E+09,9E+09,9E+09,9E+09,9E+09,9E+09]];

    CONST robtarget rA_t337 := [[1324.12,1324.12,2692.34],[2.37779E-6,0.141217,0.141218,0.979855],[0,-3,-1,0],[9E+09,9E+09,9E+09,9E+09,9E+09,9E+09]];
    CONST robtarget rB_t337 := [[-80.751,-1365.57,2949.42],[0.825436,0.276774,-0.134228,-0.473323],[-1,-2,2,0],[9E+09,9E+09,9E+09,9E+09,9E+09,9E+09]];
    CONST robtarget rB_t337_c2 := [[-80.751,-1365.57,2949.42],[0.825436,0.276774,-0.134228,-0.473323],[0,0,-4,0],[9E+09,9E+09,9E+09,9E+09,9E+09,9E+09]];
    CONST robtarget rB_t337_c5 := [[-80.751,-1365.57,2949.42],[0.825436,0.276774,-0.134228,-0.473323],[0,0,0,0],[9E+09,9E+09,9E+09,9E+09,9E+09,9E+09]];
    CONST jointtarget jA_t337 := [[44.9999,6.24592,-27.8326,-180,45.3731,-45.0001],[9E+09,9E+09,9E+09,9E+09,9E+09,9E+09]];
    CONST jointtarget jB_t337 := [[-89.9995,-8.97794,-25.345,-135,43.1501,180],[9E+09,9E+09,9E+09,9E+09,9E+09,9E+09]];
    CONST jointtarget jBseed_t337 := [[-89.9995,-8.97794,-25.345,-135,43.1501,180],[9E+09,9E+09,9E+09,9E+09,9E+09,9E+09]];

    CONST robtarget rA_t338 := [[-80.751,-1365.57,2949.42],[0.825436,0.276774,-0.134228,-0.473323],[-1,-2,2,0],[9E+09,9E+09,9E+09,9E+09,9E+09,9E+09]];
    CONST robtarget rB_t338 := [[1914.76,1935.69,646.87],[0.039023,-0.590297,-0.620247,-0.515093],[0,1,4,0],[9E+09,9E+09,9E+09,9E+09,9E+09,9E+09]];
    CONST robtarget rB_t338_c4 := [[1914.76,1935.69,646.87],[0.039023,-0.590297,-0.620247,-0.515093],[0,-4,0,0],[9E+09,9E+09,9E+09,9E+09,9E+09,9E+09]];
    CONST robtarget rB_t338_c7 := [[1914.76,1935.69,646.87],[0.039023,-0.590297,-0.620247,-0.515093],[0,-4,4,0],[9E+09,9E+09,9E+09,9E+09,9E+09,9E+09]];
    CONST jointtarget jA_t338 := [[-89.9995,-8.97794,-25.345,-135,43.1501,180],[9E+09,9E+09,9E+09,9E+09,9E+09,9E+09]];
    CONST jointtarget jB_t338 := [[45,49.3027,-16.2835,135,7.19993,360],[9E+09,9E+09,9E+09,9E+09,9E+09,9E+09]];
    CONST jointtarget jBseed_t338 := [[45,49.3027,-16.2835,135,7.19993,360],[9E+09,9E+09,9E+09,9E+09,9E+09,9E+09]];

    CONST robtarget rA_t339 := [[1914.76,1935.69,646.87],[0.039023,-0.590297,-0.620247,-0.515093],[0,1,4,0],[9E+09,9E+09,9E+09,9E+09,9E+09,9E+09]];
    CONST robtarget rB_t339 := [[-1543.09,1400.58,2439.78],[0.114741,-0.621638,-0.0185312,0.774633],[1,0,-2,0],[9E+09,9E+09,9E+09,9E+09,9E+09,9E+09]];
    CONST robtarget rB_t339_c8 := [[-1543.09,1400.58,2439.78],[0.114741,-0.621638,-0.0185312,0.774633],[0,0,4,0],[9E+09,9E+09,9E+09,9E+09,9E+09,9E+09]];
    CONST jointtarget jA_t339 := [[45,49.3027,-16.2835,135,7.19993,360],[9E+09,9E+09,9E+09,9E+09,9E+09,9E+09]];
    CONST jointtarget jB_t339 := [[135,10.6406,-27.1383,89.9999,37.1166,-90.0001],[9E+09,9E+09,9E+09,9E+09,9E+09,9E+09]];
    CONST jointtarget jBseed_t339 := [[135,10.6406,-27.1383,89.9999,37.1166,-90.0001],[9E+09,9E+09,9E+09,9E+09,9E+09,9E+09]];

    CONST robtarget rA_t340 := [[-1543.09,1400.58,2439.78],[0.114741,-0.621638,-0.0185312,0.774633],[1,0,-2,0],[9E+09,9E+09,9E+09,9E+09,9E+09,9E+09]];
    CONST robtarget rB_t340 := [[1773.81,1649.19,1063.96],[0.0372455,-0.654581,-0.115948,-0.746118],[0,2,-1,0],[9E+09,9E+09,9E+09,9E+09,9E+09,9E+09]];
    CONST robtarget rB_t340_c5 := [[1773.81,1649.19,1063.96],[0.0372455,-0.654581,-0.115948,-0.746118],[0,0,0,0],[9E+09,9E+09,9E+09,9E+09,9E+09,9E+09]];
    CONST robtarget rB_t340_c6 := [[1773.81,1649.19,1063.96],[0.0372455,-0.654581,-0.115948,-0.746118],[0,4,0,0],[9E+09,9E+09,9E+09,9E+09,9E+09,9E+09]];
    CONST jointtarget jA_t340 := [[135,10.6406,-27.1383,89.9999,37.1166,-90.0001],[9E+09,9E+09,9E+09,9E+09,9E+09,9E+09]];
    CONST jointtarget jB_t340 := [[45.0005,27.9885,2.56569,225,48.2772,-44.9995],[9E+09,9E+09,9E+09,9E+09,9E+09,9E+09]];
    CONST jointtarget jBseed_t340 := [[45.0005,27.9885,2.56569,225,48.2772,-44.9995],[9E+09,9E+09,9E+09,9E+09,9E+09,9E+09]];

    CONST robtarget rA_t341 := [[1773.81,1649.19,1063.96],[0.0372455,-0.654581,-0.115948,-0.746118],[0,2,-1,0],[9E+09,9E+09,9E+09,9E+09,9E+09,9E+09]];
    CONST robtarget rB_t341 := [[-766.297,661.309,2194.42],[0.12832,-0.740678,0.0947186,0.652655],[1,0,3,0],[9E+09,9E+09,9E+09,9E+09,9E+09,9E+09]];
    CONST robtarget rB_t341_c5 := [[-766.297,661.309,2194.42],[0.12832,-0.740678,0.0947186,0.652655],[0,0,0,0],[9E+09,9E+09,9E+09,9E+09,9E+09,9E+09]];
    CONST jointtarget jA_t341 := [[45.0005,27.9885,2.56569,225,48.2772,-44.9995],[9E+09,9E+09,9E+09,9E+09,9E+09,9E+09]];
    CONST jointtarget jB_t341 := [[134.999,-46.5963,24.2198,44.9991,38.9624,314.999],[9E+09,9E+09,9E+09,9E+09,9E+09,9E+09]];
    CONST jointtarget jBseed_t341 := [[134.999,-46.5963,24.2198,44.9991,38.9624,314.999],[9E+09,9E+09,9E+09,9E+09,9E+09,9E+09]];

    CONST robtarget rA_t342 := [[-766.297,661.309,2194.42],[0.12832,-0.740678,0.0947186,0.652655],[1,0,3,0],[9E+09,9E+09,9E+09,9E+09,9E+09,9E+09]];
    CONST robtarget rB_t342 := [[-1404.87,1257.19,37.0505],[0.183196,-0.609015,-0.699961,0.324952],[1,1,1,0],[9E+09,9E+09,9E+09,9E+09,9E+09,9E+09]];
    CONST robtarget rB_t342_c5 := [[-1404.87,1257.19,37.0505],[0.183196,-0.609015,-0.699961,0.324952],[0,0,0,0],[9E+09,9E+09,9E+09,9E+09,9E+09,9E+09]];
    CONST jointtarget jA_t342 := [[134.999,-46.5963,24.2198,44.9991,38.9624,314.999],[9E+09,9E+09,9E+09,9E+09,9E+09,9E+09]];
    CONST jointtarget jB_t342 := [[135.001,41.2384,26.3701,90.001,38.6895,135.001],[9E+09,9E+09,9E+09,9E+09,9E+09,9E+09]];
    CONST jointtarget jBseed_t342 := [[135.001,41.2384,26.3701,90.001,38.6895,135.001],[9E+09,9E+09,9E+09,9E+09,9E+09,9E+09]];

    CONST robtarget rA_t344 := [[919.116,-818.836,2400.69],[0.55952,-0.186649,0.70986,-0.384965],[-1,0,-1,0],[9E+09,9E+09,9E+09,9E+09,9E+09,9E+09]];
    CONST robtarget rB_t344 := [[1320.22,1320.24,437.708],[0.060526,0.912251,0.377864,-0.146127],[0,0,2,0],[9E+09,9E+09,9E+09,9E+09,9E+09,9E+09]];
    CONST robtarget rB_t344_c2 := [[1320.22,1320.24,437.708],[0.060526,0.912251,0.377864,-0.146127],[0,0,-4,0],[9E+09,9E+09,9E+09,9E+09,9E+09,9E+09]];
    CONST robtarget rB_t344_c5 := [[1320.22,1320.24,437.708],[0.060526,0.912251,0.377864,-0.146127],[0,0,0,0],[9E+09,9E+09,9E+09,9E+09,9E+09,9E+09]];
    CONST jointtarget jA_t344 := [[-44.9995,-31.6288,8.57631,45.0005,36.8969,-89.9995],[9E+09,9E+09,9E+09,9E+09,9E+09,9E+09]];
    CONST jointtarget jB_t344 := [[45.0005,25.3151,26.1599,0.000467155,56.726,180],[9E+09,9E+09,9E+09,9E+09,9E+09,9E+09]];
    CONST jointtarget jBseed_t344 := [[45.0005,25.3151,26.1599,0.000467391,56.726,180],[9E+09,9E+09,9E+09,9E+09,9E+09,9E+09]];

    CONST robtarget rA_t345 := [[1320.22,1320.24,437.708],[0.060526,0.912251,0.377864,-0.146127],[0,0,2,0],[9E+09,9E+09,9E+09,9E+09,9E+09,9E+09]];
    CONST robtarget rB_t345 := [[-0.0131098,-1420.93,3172.78],[0.959876,0.280425,2.28888E-6,-1.33506E-5],[-2,1,-2,0],[9E+09,9E+09,9E+09,9E+09,9E+09,9E+09]];
    CONST robtarget rB_t345_c7 := [[-0.0131098,-1420.93,3172.78],[0.959876,0.280425,2.28888E-6,-1.33506E-5],[0,-4,4,0],[9E+09,9E+09,9E+09,9E+09,9E+09,9E+09]];
    CONST jointtarget jA_t345 := [[45.0005,25.3151,26.1599,0.000467155,56.726,180],[9E+09,9E+09,9E+09,9E+09,9E+09,9E+09]];
    CONST jointtarget jB_t345 := [[-90.0005,3.55052,-49.0661,179.999,11.9132,-90.0005],[9E+09,9E+09,9E+09,9E+09,9E+09,9E+09]];
    CONST jointtarget jBseed_t345 := [[-90.0005,3.55052,-49.0661,179.999,11.9132,-90.0005],[9E+09,9E+09,9E+09,9E+09,9E+09,9E+09]];

    CONST robtarget rA_t346 := [[-0.0131098,-1420.93,3172.78],[0.959876,0.280425,2.28888E-6,-1.33506E-5],[-2,1,-2,0],[9E+09,9E+09,9E+09,9E+09,9E+09,9E+09]];
    CONST robtarget rB_t346 := [[1569.04,28.9036,1598.31],[0.206548,0.632154,0.322141,0.673754],[0,-3,0,0],[9E+09,9E+09,9E+09,9E+09,9E+09,9E+09]];
    CONST robtarget rB_t346_c2 := [[1569.04,28.9036,1598.31],[0.206548,0.632154,0.322141,0.673754],[0,0,-4,0],[9E+09,9E+09,9E+09,9E+09,9E+09,9E+09]];
    CONST robtarget rB_t346_c5 := [[1569.04,28.9036,1598.31],[0.206548,0.632154,0.322141,0.673754],[0,0,0,0],[9E+09,9E+09,9E+09,9E+09,9E+09,9E+09]];
    CONST jointtarget jA_t346 := [[-90.0005,3.55052,-49.0661,179.999,11.9132,-90.0005],[9E+09,9E+09,9E+09,9E+09,9E+09,9E+09]];
    CONST jointtarget jB_t346 := [[0.000866128,-25.0075,35.515,-224.999,14.1563,0.000873368],[9E+09,9E+09,9E+09,9E+09,9E+09,9E+09]];
    CONST jointtarget jBseed_t346 := [[0.000866207,-25.0075,35.515,-224.999,14.1563,0.000866207],[9E+09,9E+09,9E+09,9E+09,9E+09,9E+09]];

    CONST robtarget rA_t347 := [[1569.04,28.9036,1598.31],[0.206548,0.632154,0.322141,0.673754],[0,-3,0,0],[9E+09,9E+09,9E+09,9E+09,9E+09,9E+09]];
    CONST robtarget rB_t347 := [[1070.92,-930.997,1731.79],[0.0863215,0.487771,0.0394632,0.867797],[-1,-3,0,0],[9E+09,9E+09,9E+09,9E+09,9E+09,9E+09]];
    CONST robtarget rB_t347_c4 := [[1070.92,-930.997,1731.79],[0.0863215,0.487771,0.0394632,0.867797],[0,-4,0,0],[9E+09,9E+09,9E+09,9E+09,9E+09,9E+09]];
    CONST jointtarget jA_t347 := [[0.000866128,-25.0075,35.515,-224.999,14.1563,0.000873368],[9E+09,9E+09,9E+09,9E+09,9E+09,9E+09]];
    CONST jointtarget jB_t347 := [[-44.9991,-30.4386,37.467,-224.999,56.8944,45.0009],[9E+09,9E+09,9E+09,9E+09,9E+09,9E+09]];
    CONST jointtarget jBseed_t347 := [[-44.9991,-30.4386,37.467,-224.999,56.8944,45.0009],[9E+09,9E+09,9E+09,9E+09,9E+09,9E+09]];

    CONST robtarget rA_t350 := [[-974.253,-1082.74,-48.5458],[0.168298,0.902168,-0.351407,0.185154],[-2,-3,0,0],[9E+09,9E+09,9E+09,9E+09,9E+09,9E+09]];
    CONST robtarget rB_t350 := [[1771.06,-1607.48,2383.99],[0.617745,0.377794,0.486442,0.488915],[-1,-3,-4,0],[9E+09,9E+09,9E+09,9E+09,9E+09,9E+09]];
    CONST robtarget rB_t350_c4 := [[1771.06,-1607.48,2383.99],[0.617745,0.377794,0.486442,0.488915],[0,-4,0,0],[9E+09,9E+09,9E+09,9E+09,9E+09,9E+09]];
    CONST jointtarget jA_t350 := [[-135,35.053,44.9535,-270,27.344,5.79545E-5],[9E+09,9E+09,9E+09,9E+09,9E+09,9E+09]];
    CONST jointtarget jB_t350 := [[-44.9994,30.2335,-49.7723,-269.999,43.8258,-359.999],[9E+09,9E+09,9E+09,9E+09,9E+09,9E+09]];
    CONST jointtarget jBseed_t350 := [[-44.9994,30.2335,-49.7723,-269.999,43.8258,-359.999],[9E+09,9E+09,9E+09,9E+09,9E+09,9E+09]];

    CONST robtarget rA_t353 := [[934.182,93.6014,2972.1],[0.23936,-0.0184625,0.298568,0.923701],[0,1,0,0],[9E+09,9E+09,9E+09,9E+09,9E+09,9E+09]];
    CONST robtarget rB_t353 := [[-1429.04,1429.08,2902.01],[0.376409,-0.166895,0.0691241,0.908672],[1,1,-3,0],[9E+09,9E+09,9E+09,9E+09,9E+09,9E+09]];
    CONST robtarget rB_t353_c2 := [[-1429.04,1429.08,2902.01],[0.376409,-0.166895,0.0691241,0.908672],[0,0,-4,0],[9E+09,9E+09,9E+09,9E+09,9E+09,9E+09]];
    CONST robtarget rB_t353_c5 := [[-1429.04,1429.08,2902.01],[0.376409,-0.166895,0.0691241,0.908672],[0,0,0,0],[9E+09,9E+09,9E+09,9E+09,9E+09,9E+09]];
    CONST jointtarget jA_t353 := [[0.000774368,-24.4508,-15.4146,135.001,52.4247,0.000772327],[9E+09,9E+09,9E+09,9E+09,9E+09,9E+09]];
    CONST jointtarget jB_t353 := [[134.999,27.5747,-64.1701,179.999,32.5901,-180.001],[9E+09,9E+09,9E+09,9E+09,9E+09,9E+09]];
    CONST jointtarget jBseed_t353 := [[134.999,27.5747,-64.1701,179.999,32.5901,-180.001],[9E+09,9E+09,9E+09,9E+09,9E+09,9E+09]];

    CONST robtarget rA_t354 := [[-1429.04,1429.08,2902.01],[0.376409,-0.166895,0.0691241,0.908672],[1,1,-3,0],[9E+09,9E+09,9E+09,9E+09,9E+09,9E+09]];
    CONST robtarget rB_t354 := [[-862.14,767.479,-343.392],[0.335042,0.94133,-0.0120363,0.038729],[1,0,2,0],[9E+09,9E+09,9E+09,9E+09,9E+09,9E+09]];
    CONST robtarget rB_t354_c5 := [[-862.14,767.479,-343.392],[0.335042,0.94133,-0.0120363,0.038729],[0,0,0,0],[9E+09,9E+09,9E+09,9E+09,9E+09,9E+09]];
    CONST jointtarget jA_t354 := [[134.999,27.5747,-64.1701,179.999,32.5901,-180.001],[9E+09,9E+09,9E+09,9E+09,9E+09,9E+09]];
    CONST jointtarget jB_t354 := [[135,52.8843,43.6918,44.9999,34.5311,270],[9E+09,9E+09,9E+09,9E+09,9E+09,9E+09]];
    CONST jointtarget jBseed_t354 := [[135,52.8843,43.6918,44.9999,34.5311,270],[9E+09,9E+09,9E+09,9E+09,9E+09,9E+09]];

    CONST robtarget rA_t357 := [[49.4146,-1691.92,1555.62],[0.164153,0.345684,-0.592193,0.709129],[-1,-3,1,0],[9E+09,9E+09,9E+09,9E+09,9E+09,9E+09]];
    CONST robtarget rB_t357 := [[-1901.01,-1901.05,1493.05],[0.759341,0.52627,-0.217993,-0.314518],[-2,-2,3,0],[9E+09,9E+09,9E+09,9E+09,9E+09,9E+09]];
    CONST robtarget rB_t357_c4 := [[-1901.01,-1901.05,1493.05],[0.759341,0.52627,-0.217993,-0.314518],[0,-4,0,0],[9E+09,9E+09,9E+09,9E+09,9E+09,9E+09]];
    CONST robtarget rB_t357_c7 := [[-1901.01,-1901.05,1493.05],[0.759341,0.52627,-0.217993,-0.314518],[0,-4,4,0],[9E+09,9E+09,9E+09,9E+09,9E+09,9E+09]];
    CONST jointtarget jA_t357 := [[-89.9997,-17.4413,31.9047,-225,24.7328,90.0003],[9E+09,9E+09,9E+09,9E+09,9E+09,9E+09]];
    CONST jointtarget jB_t357 := [[-134.999,35.9905,-23.4129,-179.999,33.1284,270.001],[9E+09,9E+09,9E+09,9E+09,9E+09,9E+09]];
    CONST jointtarget jBseed_t357 := [[-134.999,35.9905,-23.4129,-179.999,33.1285,270.001],[9E+09,9E+09,9E+09,9E+09,9E+09,9E+09]];

    CONST robtarget rA_t360 := [[2836.44,55.9984,497.744],[0.503285,0.221475,0.746956,0.373779],[-1,1,2,0],[9E+09,9E+09,9E+09,9E+09,9E+09,9E+09]];
    CONST robtarget rB_t360 := [[-0.0397288,-2924.84,1144.11],[0.631603,0.317902,0.317912,-0.631623],[-2,-3,1,0],[9E+09,9E+09,9E+09,9E+09,9E+09,9E+09]];
    CONST robtarget rB_t360_c5 := [[-0.0397288,-2924.84,1144.11],[0.631603,0.317902,0.317912,-0.631623],[0,0,0,0],[9E+09,9E+09,9E+09,9E+09,9E+09,9E+09]];
    CONST jointtarget jA_t360 := [[-0.000510018,59.8352,-25.8449,134.999,28.3218,269.999],[9E+09,9E+09,9E+09,9E+09,9E+09,9E+09]];
    CONST jointtarget jB_t360 := [[-90.0008,56.1657,-39.6197,-180.001,53.1114,179.999],[9E+09,9E+09,9E+09,9E+09,9E+09,9E+09]];
    CONST jointtarget jBseed_t360 := [[-90.0008,56.1657,-39.6197,-180.001,53.1114,179.999],[9E+09,9E+09,9E+09,9E+09,9E+09,9E+09]];

    CONST robtarget rA_t361 := [[-0.0397288,-2924.84,1144.11],[0.631603,0.317902,0.317912,-0.631623],[-2,-3,1,0],[9E+09,9E+09,9E+09,9E+09,9E+09,9E+09]];
    CONST robtarget rB_t361 := [[1926.76,-1926.77,1280.3],[0.243109,-0.295541,0.713495,-0.586923],[-1,-3,-4,0],[9E+09,9E+09,9E+09,9E+09,9E+09,9E+09]];
    CONST robtarget rB_t361_c5 := [[1926.76,-1926.77,1280.3],[0.243109,-0.295541,0.713495,-0.586923],[0,0,0,0],[9E+09,9E+09,9E+09,9E+09,9E+09,9E+09]];
    CONST jointtarget jA_t361 := [[-90.0008,56.1657,-39.6197,-180.001,53.1114,179.999],[9E+09,9E+09,9E+09,9E+09,9E+09,9E+09]];
    CONST jointtarget jB_t361 := [[-45.0001,38.5614,-22.5996,-180,4.84329,-270],[9E+09,9E+09,9E+09,9E+09,9E+09,9E+09]];
    CONST jointtarget jBseed_t361 := [[-45.0001,38.5614,-22.5996,-180,4.84329,-270],[9E+09,9E+09,9E+09,9E+09,9E+09,9E+09]];

    CONST robtarget rA_t362 := [[1926.76,-1926.77,1280.3],[0.243109,-0.295541,0.713495,-0.586923],[-1,-3,-4,0],[9E+09,9E+09,9E+09,9E+09,9E+09,9E+09]];
    CONST robtarget rB_t362 := [[793.622,0.0122808,2208.73],[0.869091,0.12982,0.313397,0.360013],[0,2,2,0],[9E+09,9E+09,9E+09,9E+09,9E+09,9E+09]];
    CONST robtarget rB_t362_c4 := [[793.622,0.0122808,2208.73],[0.869091,0.12982,0.313397,0.360013],[0,-4,0,0],[9E+09,9E+09,9E+09,9E+09,9E+09,9E+09]];
    CONST jointtarget jA_t362 := [[-45.0001,38.5614,-22.5996,-180,4.84329,-270],[9E+09,9E+09,9E+09,9E+09,9E+09,9E+09]];
    CONST jointtarget jB_t362 := [[0.000975443,-58.6193,33.9796,180.001,25.7015,225.001],[9E+09,9E+09,9E+09,9E+09,9E+09,9E+09]];
    CONST jointtarget jBseed_t362 := [[0.000975585,-58.6193,33.9796,180.001,25.7015,225.001],[9E+09,9E+09,9E+09,9E+09,9E+09,9E+09]];

    CONST robtarget rA_t363 := [[793.622,0.0122808,2208.73],[0.869091,0.12982,0.313397,0.360013],[0,2,2,0],[9E+09,9E+09,9E+09,9E+09,9E+09,9E+09]];
    CONST robtarget rB_t363 := [[-1109.35,909.346,3202.63],[0.721877,-0.0538489,-0.524029,0.448762],[1,-3,-2,0],[9E+09,9E+09,9E+09,9E+09,9E+09,9E+09]];
    CONST robtarget rB_t363_c5 := [[-1109.35,909.346,3202.63],[0.721877,-0.0538489,-0.524029,0.448762],[0,0,0,0],[9E+09,9E+09,9E+09,9E+09,9E+09,9E+09]];
    CONST jointtarget jA_t363 := [[0.000975443,-58.6193,33.9796,180.001,25.7015,225.001],[9E+09,9E+09,9E+09,9E+09,9E+09,9E+09]];
    CONST jointtarget jB_t363 := [[135.001,19.7192,-76.4849,-269.999,57.8594,-179.999],[9E+09,9E+09,9E+09,9E+09,9E+09,9E+09]];
    CONST jointtarget jBseed_t363 := [[135.001,19.7192,-76.4849,-269.999,57.8594,-179.999],[9E+09,9E+09,9E+09,9E+09,9E+09,9E+09]];

    CONST robtarget rA_t364 := [[-1109.35,909.346,3202.63],[0.721877,-0.0538489,-0.524029,0.448762],[1,-3,-2,0],[9E+09,9E+09,9E+09,9E+09,9E+09,9E+09]];
    CONST robtarget rB_t364 := [[284.402,79.1335,2966.15],[0.62714,-0.135573,0.205564,0.738958],[-1,1,3,0],[9E+09,9E+09,9E+09,9E+09,9E+09,9E+09]];
    CONST robtarget rB_t364_c4 := [[284.402,79.1335,2966.15],[0.62714,-0.135573,0.205564,0.738958],[0,-4,0,0],[9E+09,9E+09,9E+09,9E+09,9E+09,9E+09]];
    CONST jointtarget jA_t364 := [[135.001,19.7192,-76.4849,-269.999,57.8594,-179.999],[9E+09,9E+09,9E+09,9E+09,9E+09,9E+09]];
    CONST jointtarget jB_t364 := [[-8.78707E-6,-45.5892,-8.11457,135,42.0771,315],[9E+09,9E+09,9E+09,9E+09,9E+09,9E+09]];
    CONST jointtarget jBseed_t364 := [[-8.94198E-6,-45.5892,-8.11457,135,42.0771,315],[9E+09,9E+09,9E+09,9E+09,9E+09,9E+09]];

    CONST robtarget rA_t368 := [[84.7731,2023.34,269.846],[0.437023,-0.250702,0.786103,0.358052],[0,-2,-3,0],[9E+09,9E+09,9E+09,9E+09,9E+09,9E+09]];
    CONST robtarget rB_t368 := [[1729.57,40.279,353.718],[0.174808,0.63068,0.674131,0.342392],[0,-3,-1,0],[9E+09,9E+09,9E+09,9E+09,9E+09,9E+09]];
    CONST robtarget rB_t368_c4 := [[1729.57,40.279,353.718],[0.174808,0.63068,0.674131,0.342392],[0,-4,0,0],[9E+09,9E+09,9E+09,9E+09,9E+09,9E+09]];
    CONST jointtarget jA_t368 := [[89.9997,35.1958,25.7115,-135,45.873,-180],[9E+09,9E+09,9E+09,9E+09,9E+09,9E+09]];
    CONST jointtarget jB_t368 := [[0.000310973,19.3603,41.5653,-225,19.939,-44.9997],[9E+09,9E+09,9E+09,9E+09,9E+09,9E+09]];
    CONST jointtarget jBseed_t368 := [[0.000310831,19.3603,41.5653,-225,19.939,-44.9997],[9E+09,9E+09,9E+09,9E+09,9E+09,9E+09]];

    CONST robtarget rA_t374 := [[-1511.52,1511.48,2706.65],[0.221773,0.311879,-0.752942,-0.535375],[1,0,1,0],[9E+09,9E+09,9E+09,9E+09,9E+09,9E+09]];
    CONST robtarget rB_t374 := [[1986.75,73.1547,2442.87],[0.17236,0.474017,0.39046,0.770156],[0,1,-4,0],[9E+09,9E+09,9E+09,9E+09,9E+09,9E+09]];
    CONST robtarget rB_t374_c5 := [[1986.75,73.1547,2442.87],[0.17236,0.474017,0.39046,0.770156],[0,0,0,0],[9E+09,9E+09,9E+09,9E+09,9E+09,9E+09]];
    CONST jointtarget jA_t374 := [[135.001,32.5114,-72.462,0.000669259,59.1211,90.0007],[9E+09,9E+09,9E+09,9E+09,9E+09,9E+09]];
    CONST jointtarget jB_t374 := [[0.000127523,4.52833,-20.3897,90.0001,25.978,-315],[9E+09,9E+09,9E+09,9E+09,9E+09,9E+09]];
    CONST jointtarget jBseed_t374 := [[0.000127537,4.52834,-20.3897,90.0001,25.978,-315],[9E+09,9E+09,9E+09,9E+09,9E+09,9E+09]];

    CONST robtarget rA_t383 := [[-102.238,545.727,3296.53],[0.878117,-0.0919626,-0.377794,-0.278792],[0,0,-3,0],[9E+09,9E+09,9E+09,9E+09,9E+09,9E+09]];
    CONST robtarget rB_t383 := [[-811.762,712.753,2438.59],[0.235641,-0.389239,-0.0371921,0.889709],[1,-3,-2,0],[9E+09,9E+09,9E+09,9E+09,9E+09,9E+09]];
    CONST robtarget rB_t383_c2 := [[-811.762,712.753,2438.59],[0.235641,-0.389239,-0.0371921,0.889709],[0,0,-4,0],[9E+09,9E+09,9E+09,9E+09,9E+09,9E+09]];
    CONST jointtarget jA_t383 := [[89.9997,-20.2869,-41.6352,89.9997,37.7502,-225],[9E+09,9E+09,9E+09,9E+09,9E+09,9E+09]];
    CONST jointtarget jB_t383 := [[135,-38.327,15.9517,-225,36.3622,-135],[9E+09,9E+09,9E+09,9E+09,9E+09,9E+09]];
    CONST jointtarget jBseed_t383 := [[135,-38.327,15.9517,-225,36.3622,-135],[9E+09,9E+09,9E+09,9E+09,9E+09,9E+09]];

    CONST robtarget rA_t389 := [[-1920.24,2018.01,1925.44],[0.142011,-0.206171,0.439219,0.862794],[1,2,-2,0],[9E+09,9E+09,9E+09,9E+09,9E+09,9E+09]];
    CONST robtarget rB_t389 := [[2676.14,94.0751,955.136],[0.536479,-0.68276,0.460651,-0.183928],[0,-3,2,0],[9E+09,9E+09,9E+09,9E+09,9E+09,9E+09]];
    CONST robtarget rB_t389_c5 := [[2676.14,94.0751,955.136],[0.536479,-0.68276,0.460651,-0.183928],[0,0,0,0],[9E+09,9E+09,9E+09,9E+09,9E+09,9E+09]];
    CONST jointtarget jA_t389 := [[135,48.5958,-57.0882,225,35.8348,-180],[9E+09,9E+09,9E+09,9E+09,9E+09,9E+09]];
    CONST jointtarget jB_t389 := [[0.000768794,42.0002,-16.4263,-269.999,34.2711,180.001],[9E+09,9E+09,9E+09,9E+09,9E+09,9E+09]];
    CONST jointtarget jBseed_t389 := [[0.000768792,42.0002,-16.4263,-269.999,34.2711,180.001],[9E+09,9E+09,9E+09,9E+09,9E+09,9E+09]];

    CONST robtarget rA_t392 := [[1067.16,-0.0138624,2866.91],[0.379606,-0.116604,0.0482931,-0.916499],[-1,-3,0,0],[9E+09,9E+09,9E+09,9E+09,9E+09,9E+09]];
    CONST robtarget rB_t392 := [[15.3167,710.339,3187.43],[0.882396,-0.268231,-0.0639084,-0.381241],[1,2,0,0],[9E+09,9E+09,9E+09,9E+09,9E+09,9E+09]];
    CONST robtarget rB_t392_c2 := [[15.3167,710.339,3187.43],[0.882396,-0.268231,-0.0639084,-0.381241],[0,0,-4,0],[9E+09,9E+09,9E+09,9E+09,9E+09,9E+09]];
    CONST robtarget rB_t392_c5 := [[15.3167,710.339,3187.43],[0.882396,-0.268231,-0.0639084,-0.381241],[0,0,0,0],[9E+09,9E+09,9E+09,9E+09,9E+09,9E+09]];
    CONST jointtarget jA_t392 := [[-0.000830626,-25.0807,-8.41609,-180.001,42.002,44.9992],[9E+09,9E+09,9E+09,9E+09,9E+09,9E+09]];
    CONST jointtarget jB_t392 := [[90.0003,-24.601,-28.4912,225,7.45445,0.000298365],[9E+09,9E+09,9E+09,9E+09,9E+09,9E+09]];
    CONST jointtarget jBseed_t392 := [[90.0003,-24.601,-28.4912,225,7.45445,0.000307047],[9E+09,9E+09,9E+09,9E+09,9E+09,9E+09]];

    CONST robtarget rA_t393 := [[15.3167,710.339,3187.43],[0.882396,-0.268231,-0.0639084,-0.381241],[1,2,0,0],[9E+09,9E+09,9E+09,9E+09,9E+09,9E+09]];
    CONST robtarget rB_t393 := [[-85.9506,2650.23,1955.45],[0.596243,-0.669059,0.061531,0.439395],[1,-3,2,0],[9E+09,9E+09,9E+09,9E+09,9E+09,9E+09]];
    CONST robtarget rB_t393_c5 := [[-85.9506,2650.23,1955.45],[0.596243,-0.669059,0.061531,0.439395],[0,0,0,0],[9E+09,9E+09,9E+09,9E+09,9E+09,9E+09]];
    CONST robtarget rB_t393_c8 := [[-85.9506,2650.23,1955.45],[0.596243,-0.669059,0.061531,0.439395],[0,0,4,0],[9E+09,9E+09,9E+09,9E+09,9E+09,9E+09]];
    CONST jointtarget jA_t393 := [[90.0003,-24.601,-28.4912,225,7.45445,0.000298365],[9E+09,9E+09,9E+09,9E+09,9E+09,9E+09]];
    CONST jointtarget jB_t393 := [[90.0003,36.939,-43.4443,-270,30.9696,225],[9E+09,9E+09,9E+09,9E+09,9E+09,9E+09]];
    CONST jointtarget jBseed_t393 := [[90.0003,36.939,-43.4443,-270,30.9696,225],[9E+09,9E+09,9E+09,9E+09,9E+09,9E+09]];

    CONST robtarget rA_t394 := [[-85.9506,2650.23,1955.45],[0.596243,-0.669059,0.061531,0.439395],[1,-3,2,0],[9E+09,9E+09,9E+09,9E+09,9E+09,9E+09]];
    CONST robtarget rB_t394 := [[1237.78,115.728,1541.33],[0.247593,0.305891,0.662348,0.637514],[-1,0,3,0],[9E+09,9E+09,9E+09,9E+09,9E+09,9E+09]];
    CONST robtarget rB_t394_c7 := [[1237.78,115.728,1541.33],[0.247593,0.305891,0.662348,0.637514],[0,-4,4,0],[9E+09,9E+09,9E+09,9E+09,9E+09,9E+09]];
    CONST jointtarget jA_t394 := [[90.0003,36.939,-43.4443,-270,30.9696,225],[9E+09,9E+09,9E+09,9E+09,9E+09,9E+09]];
    CONST jointtarget jB_t394 := [[-0.000493266,-42.8242,47.9608,89.9995,43.8716,360],[9E+09,9E+09,9E+09,9E+09,9E+09,9E+09]];
    CONST jointtarget jBseed_t394 := [[-0.000492966,-42.8242,47.9608,89.9995,43.8716,360],[9E+09,9E+09,9E+09,9E+09,9E+09,9E+09]];

    CONST robtarget rA_t396 := [[-431.431,523.46,2441.2],[0.732231,-0.280709,0.178527,0.594279],[1,-2,-3,0],[9E+09,9E+09,9E+09,9E+09,9E+09,9E+09]];
    CONST robtarget rB_t396 := [[1325.12,1364.86,3005.43],[0.915051,-0.333711,0.224059,0.0334189],[0,-4,-2,0],[9E+09,9E+09,9E+09,9E+09,9E+09,9E+09]];
    CONST robtarget rB_t396_c7 := [[1325.12,1364.86,3005.43],[0.915051,-0.333711,0.224059,0.0334189],[0,-4,4,0],[9E+09,9E+09,9E+09,9E+09,9E+09,9E+09]];
    CONST jointtarget jA_t396 := [[135,-55.338,22.6447,-135,33.4416,-270],[9E+09,9E+09,9E+09,9E+09,9E+09,9E+09]];
    CONST jointtarget jB_t396 := [[45,25.0807,-68.4469,-270,9.68658,-135],[9E+09,9E+09,9E+09,9E+09,9E+09,9E+09]];
    CONST jointtarget jBseed_t396 := [[45,25.0807,-68.4469,-270,9.68657,-135],[9E+09,9E+09,9E+09,9E+09,9E+09,9E+09]];

    CONST robtarget rA_t397 := [[1325.12,1364.86,3005.43],[0.915051,-0.333711,0.224059,0.0334189],[0,-4,-2,0],[9E+09,9E+09,9E+09,9E+09,9E+09,9E+09]];
    CONST robtarget rB_t397 := [[41.4855,-161.608,3341.08],[0.032164,0.075762,-0.463803,0.882107],[-1,-1,2,0],[9E+09,9E+09,9E+09,9E+09,9E+09,9E+09]];
    CONST robtarget rB_t397_c5 := [[41.4855,-161.608,3341.08],[0.032164,0.075762,-0.463803,0.882107],[0,0,0,0],[9E+09,9E+09,9E+09,9E+09,9E+09,9E+09]];
    CONST jointtarget jA_t397 := [[45,25.0807,-68.4469,-270,9.68658,-135],[9E+09,9E+09,9E+09,9E+09,9E+09,9E+09]];
    CONST jointtarget jB_t397 := [[-45.0003,-23.6378,-52.9939,-45.0003,45.9957,270],[9E+09,9E+09,9E+09,9E+09,9E+09,9E+09]];
    CONST jointtarget jBseed_t397 := [[-45.0003,-23.6378,-52.9939,-45.0003,45.9957,270],[9E+09,9E+09,9E+09,9E+09,9E+09,9E+09]];

    CONST robtarget rA_t398 := [[41.4855,-161.608,3341.08],[0.032164,0.075762,-0.463803,0.882107],[-1,-1,2,0],[9E+09,9E+09,9E+09,9E+09,9E+09,9E+09]];
    CONST robtarget rB_t398 := [[86.685,2548.54,225.229],[0.600836,-0.468171,0.607465,0.225382],[0,2,1,0],[9E+09,9E+09,9E+09,9E+09,9E+09,9E+09]];
    CONST robtarget rB_t398_c4 := [[86.685,2548.54,225.229],[0.600836,-0.468171,0.607465,0.225382],[0,-4,0,0],[9E+09,9E+09,9E+09,9E+09,9E+09,9E+09]];
    CONST jointtarget jA_t398 := [[-45.0003,-23.6378,-52.9939,-45.0003,45.9957,270],[9E+09,9E+09,9E+09,9E+09,9E+09,9E+09]];
    CONST jointtarget jB_t398 := [[89.9995,55.9423,-6.65456,224.999,47.2134,134.999],[9E+09,9E+09,9E+09,9E+09,9E+09,9E+09]];
    CONST jointtarget jBseed_t398 := [[89.9995,55.9423,-6.65456,224.999,47.2134,134.999],[9E+09,9E+09,9E+09,9E+09,9E+09,9E+09]];

    CONST robtarget rA_t399 := [[86.685,2548.54,225.229],[0.600836,-0.468171,0.607465,0.225382],[0,2,1,0],[9E+09,9E+09,9E+09,9E+09,9E+09,9E+09]];
    CONST robtarget rB_t399 := [[1129.25,-1129.27,2978.38],[0.686444,0.240044,4.08915E-6,0.686421],[-1,-3,3,0],[9E+09,9E+09,9E+09,9E+09,9E+09,9E+09]];
    CONST robtarget rB_t399_c8 := [[1129.25,-1129.27,2978.38],[0.686444,0.240044,4.08915E-6,0.686421],[0,0,4,0],[9E+09,9E+09,9E+09,9E+09,9E+09,9E+09]];
    CONST jointtarget jA_t399 := [[89.9995,55.9423,-6.65456,224.999,47.2134,134.999],[9E+09,9E+09,9E+09,9E+09,9E+09,9E+09]];
    CONST jointtarget jB_t399 := [[-45.0007,1.8952,-36.3903,-180.001,27.7267,314.999],[9E+09,9E+09,9E+09,9E+09,9E+09,9E+09]];
    CONST jointtarget jBseed_t399 := [[-45.0007,1.8952,-36.3903,-180.001,27.7267,314.999],[9E+09,9E+09,9E+09,9E+09,9E+09,9E+09]];

    CONST robtarget rA_t402 := [[-832.618,-969.982,1856.99],[0.324405,0.545685,-0.677678,0.371136],[-2,0,1,0],[9E+09,9E+09,9E+09,9E+09,9E+09,9E+09]];
    CONST robtarget rB_t402 := [[-635.888,-665.143,3243.13],[0.864052,0.363814,-0.08678,-0.336932],[-2,0,0,0],[9E+09,9E+09,9E+09,9E+09,9E+09,9E+09]];
    CONST robtarget rB_t402_c5 := [[-635.888,-665.143,3243.13],[0.864052,0.363814,-0.08678,-0.336932],[0,0,0,0],[9E+09,9E+09,9E+09,9E+09,9E+09,9E+09]];
    CONST jointtarget jA_t402 := [[-134.999,-36.4849,30.0439,45.0006,55.327,135.001],[9E+09,9E+09,9E+09,9E+09,9E+09,9E+09]];
    CONST jointtarget jB_t402 := [[-134.999,-13.8926,-39.8102,45.0006,10.0839,45.0007],[9E+09,9E+09,9E+09,9E+09,9E+09,9E+09]];
    CONST jointtarget jBseed_t402 := [[-134.999,-13.8926,-39.8102,45.0007,10.0839,45.0007],[9E+09,9E+09,9E+09,9E+09,9E+09,9E+09]];

    CONST robtarget rA_t404 := [[-1552.06,1552.08,1866.86],[0.332459,-0.457561,0.189526,0.802614],[1,1,-3,0],[9E+09,9E+09,9E+09,9E+09,9E+09,9E+09]];
    CONST robtarget rB_t404 := [[-56.959,1973.89,1680.26],[0.740668,-0.552237,-0.348349,-0.158425],[1,-3,1,0],[9E+09,9E+09,9E+09,9E+09,9E+09,9E+09]];
    CONST robtarget rB_t404_c2 := [[-56.959,1973.89,1680.26],[0.740668,-0.552237,-0.348349,-0.158425],[0,0,-4,0],[9E+09,9E+09,9E+09,9E+09,9E+09,9E+09]];
    CONST robtarget rB_t404_c5 := [[-56.959,1973.89,1680.26],[0.740668,-0.552237,-0.348349,-0.158425],[0,0,0,0],[9E+09,9E+09,9E+09,9E+09,9E+09,9E+09]];
    CONST jointtarget jA_t404 := [[135,8.77651,-1.59215,180,37.8106,-180],[9E+09,9E+09,9E+09,9E+09,9E+09,9E+09]];
    CONST jointtarget jB_t404 := [[90.0001,-2.85836,15.1106,-225,28.8363,90.0001],[9E+09,9E+09,9E+09,9E+09,9E+09,9E+09]];
    CONST jointtarget jBseed_t404 := [[90.0001,-2.85836,15.1106,-225,28.8363,90.0001],[9E+09,9E+09,9E+09,9E+09,9E+09,9E+09]];

    CONST robtarget rA_t405 := [[-56.959,1973.89,1680.26],[0.740668,-0.552237,-0.348349,-0.158425],[1,-3,1,0],[9E+09,9E+09,9E+09,9E+09,9E+09,9E+09]];
    CONST robtarget rB_t405 := [[1414.45,-40.9812,2868.33],[0.616404,0.479359,0.323317,0.534534],[-1,-1,1,0],[9E+09,9E+09,9E+09,9E+09,9E+09,9E+09]];
    CONST robtarget rB_t405_c5 := [[1414.45,-40.9812,2868.33],[0.616404,0.479359,0.323317,0.534534],[0,0,0,0],[9E+09,9E+09,9E+09,9E+09,9E+09,9E+09]];
    CONST jointtarget jA_t405 := [[90.0001,-2.85836,15.1106,-225,28.8363,90.0001],[9E+09,9E+09,9E+09,9E+09,9E+09,9E+09]];
    CONST jointtarget jB_t405 := [[-0.000662186,-11.1789,-23.4645,-45.0007,20.2979,134.999],[9E+09,9E+09,9E+09,9E+09,9E+09,9E+09]];
    CONST jointtarget jBseed_t405 := [[-0.000662038,-11.1789,-23.4645,-45.0007,20.2979,134.999],[9E+09,9E+09,9E+09,9E+09,9E+09,9E+09]];

    CONST robtarget rA_t406 := [[1414.45,-40.9812,2868.33],[0.616404,0.479359,0.323317,0.534534],[-1,-1,1,0],[9E+09,9E+09,9E+09,9E+09,9E+09,9E+09]];
    CONST robtarget rB_t406 := [[-865.919,901.13,3122],[0.838449,-0.211363,-0.330131,-0.378607],[1,3,-1,0],[9E+09,9E+09,9E+09,9E+09,9E+09,9E+09]];
    CONST robtarget rB_t406_c5 := [[-865.919,901.13,3122],[0.838449,-0.211363,-0.330131,-0.378607],[0,0,0,0],[9E+09,9E+09,9E+09,9E+09,9E+09,9E+09]];
    CONST robtarget rB_t406_c8 := [[-865.919,901.13,3122],[0.838449,-0.211363,-0.330131,-0.378607],[0,0,4,0],[9E+09,9E+09,9E+09,9E+09,9E+09,9E+09]];
    CONST jointtarget jA_t406 := [[-0.000662186,-11.1789,-23.4645,-45.0007,20.2979,134.999],[9E+09,9E+09,9E+09,9E+09,9E+09,9E+09]];
    CONST jointtarget jB_t406 := [[135,-7.83167,-36.6362,270,8.57509,-89.9999],[9E+09,9E+09,9E+09,9E+09,9E+09,9E+09]];
    CONST jointtarget jBseed_t406 := [[135,-7.83166,-36.6362,270,8.57509,-89.9999],[9E+09,9E+09,9E+09,9E+09,9E+09,9E+09]];

    CONST robtarget rA_t408 := [[1837.97,-1944.27,1373.23],[0.190966,0.327644,-0.531303,0.757561],[-1,-2,4,0],[9E+09,9E+09,9E+09,9E+09,9E+09,9E+09]];
    CONST robtarget rB_t408 := [[-58.933,-1733.72,2638.49],[0.184483,0.39953,0.561291,-0.700924],[-1,-1,0,0],[9E+09,9E+09,9E+09,9E+09,9E+09,9E+09]];
    CONST robtarget rB_t408_c5 := [[-58.933,-1733.72,2638.49],[0.184483,0.39953,0.561291,-0.700924],[0,0,0,0],[9E+09,9E+09,9E+09,9E+09,9E+09,9E+09]];
    CONST jointtarget jA_t408 := [[-44.9997,36.5581,-20.596,-135,39.541,360],[9E+09,9E+09,9E+09,9E+09,9E+09,9E+09]];
    CONST jointtarget jB_t408 := [[-89.9995,-2.884,-22.3853,-44.9994,29.9478,0.00054559],[9E+09,9E+09,9E+09,9E+09,9E+09,9E+09]];
    CONST jointtarget jBseed_t408 := [[-89.9995,-2.884,-22.3853,-44.9994,29.9478,0.000552721],[9E+09,9E+09,9E+09,9E+09,9E+09,9E+09]];

    CONST robtarget rA_t409 := [[-58.933,-1733.72,2638.49],[0.184483,0.39953,0.561291,-0.700924],[-1,-1,0,0],[9E+09,9E+09,9E+09,9E+09,9E+09,9E+09]];
    CONST robtarget rB_t409 := [[-138.545,-2233.26,732.353],[0.427033,-0.195795,-0.802451,0.36794],[-2,2,-5,0],[9E+09,9E+09,9E+09,9E+09,9E+09,9E+09]];
    CONST robtarget rB_t409_c5 := [[-138.545,-2233.26,732.353],[0.427033,-0.195795,-0.802451,0.36794],[0,0,0,0],[9E+09,9E+09,9E+09,9E+09,9E+09,9E+09]];
    CONST robtarget rB_t409_c8 := [[-138.545,-2233.26,732.353],[0.427033,-0.195795,-0.802451,0.36794],[0,0,4,0],[9E+09,9E+09,9E+09,9E+09,9E+09,9E+09]];
    CONST jointtarget jA_t409 := [[-89.9995,-2.884,-22.3853,-44.9994,29.9478,0.00054559],[9E+09,9E+09,9E+09,9E+09,9E+09,9E+09]];
    CONST jointtarget jB_t409 := [[-90.0008,28.7942,11.9407,269.999,56.0393,-360.001],[9E+09,9E+09,9E+09,9E+09,9E+09,9E+09]];
    CONST jointtarget jBseed_t409 := [[-90.0008,28.7942,11.9407,269.999,56.0393,-360.001],[9E+09,9E+09,9E+09,9E+09,9E+09,9E+09]];

    CONST robtarget rA_t411 := [[-1065.64,931.409,-331.742],[0.209596,0.954687,0.000368102,-0.211287],[1,-3,-2,0],[9E+09,9E+09,9E+09,9E+09,9E+09,9E+09]];
    CONST robtarget rB_t411 := [[-10.1008,1466.94,43.1946],[0.128089,-0.914249,0.374724,0.0855814],[0,-3,-3,0],[9E+09,9E+09,9E+09,9E+09,9E+09,9E+09]];
    CONST robtarget rB_t411_c1 := [[-10.1008,1466.94,43.1946],[0.128089,-0.914249,0.374724,0.0855814],[0,-4,-4,0],[9E+09,9E+09,9E+09,9E+09,9E+09,9E+09]];
    CONST jointtarget jA_t411 := [[135.001,52.4448,37.4114,-269.999,34.6281,-134.999],[9E+09,9E+09,9E+09,9E+09,9E+09,9E+09]];
    CONST jointtarget jB_t411 := [[90,28.2888,47.7941,-225,4.90738,-180],[9E+09,9E+09,9E+09,9E+09,9E+09,9E+09]];
    CONST jointtarget jBseed_t411 := [[90,28.2888,47.7941,-225,4.90738,-180],[9E+09,9E+09,9E+09,9E+09,9E+09,9E+09]];

    CONST robtarget rA_t413 := [[-70.7229,-2239.45,-140.534],[0.298013,0.855281,-0.410854,-0.104318],[-2,2,2,0],[9E+09,9E+09,9E+09,9E+09,9E+09,9E+09]];
    CONST robtarget rB_t413 := [[1273.4,-1403.87,61.7876],[0.110289,0.0530668,0.834458,-0.537308],[-1,2,-3,0],[9E+09,9E+09,9E+09,9E+09,9E+09,9E+09]];
    CONST robtarget rB_t413_c6 := [[1273.4,-1403.87,61.7876],[0.110289,0.0530668,0.834458,-0.537308],[0,4,0,0],[9E+09,9E+09,9E+09,9E+09,9E+09,9E+09]];
    CONST jointtarget jA_t413 := [[-90.0007,57.7844,4.30738,269.999,25.0441,224.999],[9E+09,9E+09,9E+09,9E+09,9E+09,9E+09]];
    CONST jointtarget jB_t413 := [[-44.9995,41.0297,29.0362,225,51.3883,-270],[9E+09,9E+09,9E+09,9E+09,9E+09,9E+09]];
    CONST jointtarget jBseed_t413 := [[-44.9995,41.0297,29.0362,225,51.3883,-270],[9E+09,9E+09,9E+09,9E+09,9E+09,9E+09]];

    CONST robtarget rA_t414 := [[1273.4,-1403.87,61.7876],[0.110289,0.0530668,0.834458,-0.537308],[-1,2,-3,0],[9E+09,9E+09,9E+09,9E+09,9E+09,9E+09]];
    CONST robtarget rB_t414 := [[40.7486,-1443.03,2522.77],[0.0711807,-0.101411,0.464164,-0.877041],[-1,-3,1,0],[9E+09,9E+09,9E+09,9E+09,9E+09,9E+09]];
    CONST robtarget rB_t414_c2 := [[40.7486,-1443.03,2522.77],[0.0711807,-0.101411,0.464164,-0.877041],[0,0,-4,0],[9E+09,9E+09,9E+09,9E+09,9E+09,9E+09]];
    CONST jointtarget jA_t414 := [[-44.9995,41.0297,29.0362,225,51.3883,-270],[9E+09,9E+09,9E+09,9E+09,9E+09,9E+09]];
    CONST jointtarget jB_t414 := [[-89.9997,-20.8069,0.931105,-225,20.1825,135],[9E+09,9E+09,9E+09,9E+09,9E+09,9E+09]];
    CONST jointtarget jBseed_t414 := [[-89.9997,-20.8069,0.931122,-225,20.1825,135],[9E+09,9E+09,9E+09,9E+09,9E+09,9E+09]];

    CONST robtarget rA_t418 := [[1584.3,1575.08,1280.33],[0.392251,0.0107715,0.842364,0.369387],[0,-1,0,0],[9E+09,9E+09,9E+09,9E+09,9E+09,9E+09]];
    CONST robtarget rB_t418 := [[584.5,-597.173,3467.26],[0.374567,-0.0294507,0.140157,-0.916072],[-1,2,-4,0],[9E+09,9E+09,9E+09,9E+09,9E+09,9E+09]];
    CONST robtarget rB_t418_c4 := [[584.5,-597.173,3467.26],[0.374567,-0.0294507,0.140157,-0.916072],[0,-4,0,0],[9E+09,9E+09,9E+09,9E+09,9E+09,9E+09]];
    CONST robtarget rB_t418_c5 := [[584.5,-597.173,3467.26],[0.374567,-0.0294507,0.140157,-0.916072],[0,0,0,0],[9E+09,9E+09,9E+09,9E+09,9E+09,9E+09]];
    CONST jointtarget jA_t418 := [[44.9992,13.2627,9.32616,-45.0008,3.14768,89.9992],[9E+09,9E+09,9E+09,9E+09,9E+09,9E+09]];
    CONST jointtarget jB_t418 := [[-45.001,7.56061,-78.2979,224.999,4.34525,-315.001],[9E+09,9E+09,9E+09,9E+09,9E+09,9E+09]];
    CONST jointtarget jBseed_t418 := [[-45.001,7.56065,-78.298,224.999,4.34523,-315.001],[9E+09,9E+09,9E+09,9E+09,9E+09,9E+09]];

    CONST robtarget rA_t419 := [[584.5,-597.173,3467.26],[0.374567,-0.0294507,0.140157,-0.916072],[-1,2,-4,0],[9E+09,9E+09,9E+09,9E+09,9E+09,9E+09]];
    CONST robtarget rB_t419 := [[1372.58,1248.75,2884.68],[0.487029,0.3045,0.0786659,0.814797],[0,-2,2,0],[9E+09,9E+09,9E+09,9E+09,9E+09,9E+09]];
    CONST robtarget rB_t419_c2 := [[1372.58,1248.75,2884.68],[0.487029,0.3045,0.0786659,0.814797],[0,0,-4,0],[9E+09,9E+09,9E+09,9E+09,9E+09,9E+09]];
    CONST jointtarget jA_t419 := [[-45.001,7.56061,-78.2979,224.999,4.34525,-315.001],[9E+09,9E+09,9E+09,9E+09,9E+09,9E+09]];
    CONST jointtarget jB_t419 := [[44.9992,14.8082,-47.2014,-135.001,47.8378,224.999],[9E+09,9E+09,9E+09,9E+09,9E+09,9E+09]];
    CONST jointtarget jBseed_t419 := [[44.9992,14.8082,-47.2015,-135.001,47.8378,224.999],[9E+09,9E+09,9E+09,9E+09,9E+09,9E+09]];

    CONST robtarget rA_t424 := [[-1987.08,1987.14,1751.17],[0.374042,-0.848647,-3.20923E-6,0.37402],[1,-1,3,0],[9E+09,9E+09,9E+09,9E+09,9E+09,9E+09]];
    CONST robtarget rB_t424 := [[1084.82,1172.66,1607.04],[0.639339,-0.740918,0.175007,-0.107974],[0,1,-2,0],[9E+09,9E+09,9E+09,9E+09,9E+09,9E+09]];
    CONST robtarget rB_t424_c5 := [[1084.82,1172.66,1607.04],[0.639339,-0.740918,0.175007,-0.107974],[0,0,0,0],[9E+09,9E+09,9E+09,9E+09,9E+09,9E+09]];
    CONST jointtarget jA_t424 := [[134.999,48.1234,-55.8822,-0.000908437,33.8884,314.999],[9E+09,9E+09,9E+09,9E+09,9E+09,9E+09]];
    CONST jointtarget jB_t424 := [[45.0008,-22.8724,32.7458,90.0008,21.8268,-179.999],[9E+09,9E+09,9E+09,9E+09,9E+09,9E+09]];
    CONST jointtarget jBseed_t424 := [[45.0008,-22.8724,32.7458,90.0008,21.8268,-179.999],[9E+09,9E+09,9E+09,9E+09,9E+09,9E+09]];

    CONST robtarget rA_t425 := [[1084.82,1172.66,1607.04],[0.639339,-0.740918,0.175007,-0.107974],[0,1,-2,0],[9E+09,9E+09,9E+09,9E+09,9E+09,9E+09]];
    CONST robtarget rB_t425 := [[-1855.99,1777.99,1374.25],[0.599652,0.100508,-0.682489,-0.405617],[1,-3,-4,0],[9E+09,9E+09,9E+09,9E+09,9E+09,9E+09]];
    CONST robtarget rB_t425_c5 := [[-1855.99,1777.99,1374.25],[0.599652,0.100508,-0.682489,-0.405617],[0,0,0,0],[9E+09,9E+09,9E+09,9E+09,9E+09,9E+09]];
    CONST jointtarget jA_t425 := [[45.0008,-22.8724,32.7458,90.0008,21.8268,-179.999],[9E+09,9E+09,9E+09,9E+09,9E+09,9E+09]];
    CONST jointtarget jB_t425 := [[135,29.7867,-12.2407,-225,27.8347,-360],[9E+09,9E+09,9E+09,9E+09,9E+09,9E+09]];
    CONST jointtarget jBseed_t425 := [[135,29.7867,-12.2407,-225,27.8347,-360],[9E+09,9E+09,9E+09,9E+09,9E+09,9E+09]];

    CONST robtarget rA_t426 := [[-1855.99,1777.99,1374.25],[0.599652,0.100508,-0.682489,-0.405617],[1,-3,-4,0],[9E+09,9E+09,9E+09,9E+09,9E+09,9E+09]];
    CONST robtarget rB_t426 := [[-51.914,1806.06,2728.88],[0.870514,-0.309432,-0.273699,-0.267479],[0,1,-4,0],[9E+09,9E+09,9E+09,9E+09,9E+09,9E+09]];
    CONST robtarget rB_t426_c1 := [[-51.914,1806.06,2728.88],[0.870514,-0.309432,-0.273699,-0.267479],[0,-4,-4,0],[9E+09,9E+09,9E+09,9E+09,9E+09,9E+09]];
    CONST jointtarget jA_t426 := [[135,29.7867,-12.2407,-225,27.8347,-360],[9E+09,9E+09,9E+09,9E+09,9E+09,9E+09]];
    CONST jointtarget jB_t426 := [[89.9993,2.57638,-27.3486,134.999,26.0915,-270.001],[9E+09,9E+09,9E+09,9E+09,9E+09,9E+09]];
    CONST jointtarget jBseed_t426 := [[89.9993,2.57637,-27.3486,134.999,26.0915,-270.001],[9E+09,9E+09,9E+09,9E+09,9E+09,9E+09]];

    CONST robtarget rA_t428 := [[596.717,537.394,2166.04],[0.585289,-0.423842,0.107426,-0.682828],[0,2,-1,0],[9E+09,9E+09,9E+09,9E+09,9E+09,9E+09]];
    CONST robtarget rB_t428 := [[-1114.25,1236.98,2779.88],[0.549848,-0.240739,-0.243462,-0.761865],[1,-2,2,0],[9E+09,9E+09,9E+09,9E+09,9E+09,9E+09]];
    CONST robtarget rB_t428_c5 := [[-1114.25,1236.98,2779.88],[0.549848,-0.240739,-0.243462,-0.761865],[0,0,0,0],[9E+09,9E+09,9E+09,9E+09,9E+09,9E+09]];
    CONST jointtarget jA_t428 := [[44.9992,-59.6118,34.9992,224.999,20.8014,-0.000831889],[9E+09,9E+09,9E+09,9E+09,9E+09,9E+09]];
    CONST jointtarget jB_t428 := [[134.999,-1.08951,-25.0911,-135.001,47.2903,269.999],[9E+09,9E+09,9E+09,9E+09,9E+09,9E+09]];
    CONST jointtarget jBseed_t428 := [[134.999,-1.08951,-25.0911,-135.001,47.2903,269.999],[9E+09,9E+09,9E+09,9E+09,9E+09,9E+09]];

    CONST robtarget rA_t429 := [[-1114.25,1236.98,2779.88],[0.549848,-0.240739,-0.243462,-0.761865],[1,-2,2,0],[9E+09,9E+09,9E+09,9E+09,9E+09,9E+09]];
    CONST robtarget rB_t429 := [[-1906.02,1958.88,668.612],[0.484997,-0.822663,-0.281266,0.0943042],[1,3,-4,0],[9E+09,9E+09,9E+09,9E+09,9E+09,9E+09]];
    CONST robtarget rB_t429_c8 := [[-1906.02,1958.88,668.612],[0.484997,-0.822663,-0.281266,0.0943042],[0,0,4,0],[9E+09,9E+09,9E+09,9E+09,9E+09,9E+09]];
    CONST jointtarget jA_t429 := [[134.999,-1.08951,-25.0911,-135.001,47.2903,269.999],[9E+09,9E+09,9E+09,9E+09,9E+09,9E+09]];
    CONST jointtarget jB_t429 := [[135.001,49.559,-17.8823,270.001,12.9514,-359.999],[9E+09,9E+09,9E+09,9E+09,9E+09,9E+09]];
    CONST jointtarget jBseed_t429 := [[135.001,49.559,-17.8823,270.001,12.9514,-359.999],[9E+09,9E+09,9E+09,9E+09,9E+09,9E+09]];

    CONST robtarget rA_t438 := [[-1660.44,-1567.59,512.217],[0.513309,-0.0734767,-0.820122,0.241896],[-2,2,0,0],[9E+09,9E+09,9E+09,9E+09,9E+09,9E+09]];
    CONST robtarget rB_t438 := [[-1198.87,-1198.89,1093.99],[0.650078,0.537304,-0.53731,7.07195E-6],[-2,-2,3,0],[9E+09,9E+09,9E+09,9E+09,9E+09,9E+09]];
    CONST robtarget rB_t438_c5 := [[-1198.87,-1198.89,1093.99],[0.650078,0.537304,-0.53731,7.07195E-6],[0,0,0,0],[9E+09,9E+09,9E+09,9E+09,9E+09,9E+09]];
    CONST jointtarget jA_t438 := [[-134.999,34.771,13.3332,225.001,33.7913,0.000513123],[9E+09,9E+09,9E+09,9E+09,9E+09,9E+09]];
    CONST jointtarget jB_t438 := [[-134.999,-10.6882,42.7,-179.999,23.1068,315.001],[9E+09,9E+09,9E+09,9E+09,9E+09,9E+09]];
    CONST jointtarget jBseed_t438 := [[-134.999,-10.6882,42.7,-179.999,23.1068,315.001],[9E+09,9E+09,9E+09,9E+09,9E+09,9E+09]];

    CONST robtarget rA_t440 := [[2.4233,2102.21,1285.67],[0.20665,-0.322086,-0.76724,-0.514684],[0,-2,-2,0],[9E+09,9E+09,9E+09,9E+09,9E+09,9E+09]];
    CONST robtarget rB_t440 := [[0.00603872,2841.53,1772.14],[0.863407,-0.328755,-0.136176,-0.357638],[0,1,-4,0],[9E+09,9E+09,9E+09,9E+09,9E+09,9E+09]];
    CONST robtarget rB_t440_c1 := [[0.00603872,2841.53,1772.14],[0.863407,-0.328755,-0.136176,-0.357638],[0,-4,-4,0],[9E+09,9E+09,9E+09,9E+09,9E+09,9E+09]];
    CONST robtarget rB_t440_c4 := [[0.00603872,2841.53,1772.14],[0.863407,-0.328755,-0.136176,-0.357638],[0,-4,0,0],[9E+09,9E+09,9E+09,9E+09,9E+09,9E+09]];
    CONST jointtarget jA_t440 := [[89.9997,6.60847,16.8523,-135,1.17008,-90.0003],[9E+09,9E+09,9E+09,9E+09,9E+09,9E+09]];
    CONST jointtarget jB_t440 := [[89.9999,51.3865,-54.3031,180,45.3932,-315],[9E+09,9E+09,9E+09,9E+09,9E+09,9E+09]];
    CONST jointtarget jBseed_t440 := [[89.9999,51.3865,-54.3031,180,45.3932,-315],[9E+09,9E+09,9E+09,9E+09,9E+09,9E+09]];

    CONST robtarget rA_t442 := [[1905.11,-143.228,2869],[0.0988346,-0.183969,0.55544,-0.804906],[0,3,-1,0],[9E+09,9E+09,9E+09,9E+09,9E+09,9E+09]];
    CONST robtarget rB_t442 := [[-86.0718,-2147.16,154.18],[0.499214,0.819765,-0.0694951,-0.271923],[-2,-2,2,0],[9E+09,9E+09,9E+09,9E+09,9E+09,9E+09]];
    CONST robtarget rB_t442_c5 := [[-86.0718,-2147.16,154.18],[0.499214,0.819765,-0.0694951,-0.271923],[0,0,0,0],[9E+09,9E+09,9E+09,9E+09,9E+09,9E+09]];
    CONST jointtarget jA_t442 := [[0.000702751,21.9056,-59.7424,270.001,59.0698,-44.9993],[9E+09,9E+09,9E+09,9E+09,9E+09,9E+09]];
    CONST jointtarget jB_t442 := [[-90.0009,44.051,17.2729,-135.001,46.7702,224.999],[9E+09,9E+09,9E+09,9E+09,9E+09,9E+09]];
    CONST jointtarget jBseed_t442 := [[-90.0009,44.051,17.2729,-135.001,46.7702,224.999],[9E+09,9E+09,9E+09,9E+09,9E+09,9E+09]];

    CONST robtarget rA_t443 := [[-86.0718,-2147.16,154.18],[0.499214,0.819765,-0.0694951,-0.271923],[-2,-2,2,0],[9E+09,9E+09,9E+09,9E+09,9E+09,9E+09]];
    CONST robtarget rB_t443 := [[1138.72,-1138.74,2942.88],[1.56807E-5,0.183625,-0.183619,0.965695],[-1,-3,0,0],[9E+09,9E+09,9E+09,9E+09,9E+09,9E+09]];
    CONST robtarget rB_t443_c4 := [[1138.72,-1138.74,2942.88],[1.56807E-5,0.183625,-0.183619,0.965695],[0,-4,0,0],[9E+09,9E+09,9E+09,9E+09,9E+09,9E+09]];
    CONST jointtarget jA_t443 := [[-90.0009,44.051,17.2729,-135.001,46.7702,224.999],[9E+09,9E+09,9E+09,9E+09,9E+09,9E+09]];
    CONST jointtarget jB_t443 := [[-45.0007,0.818501,-33.7202,-180.001,26.9961,44.9993],[9E+09,9E+09,9E+09,9E+09,9E+09,9E+09]];
    CONST jointtarget jBseed_t443 := [[-45.0007,0.818504,-33.7202,-180.001,26.9961,44.9993],[9E+09,9E+09,9E+09,9E+09,9E+09,9E+09]];

    CONST robtarget rA_t444 := [[1138.72,-1138.74,2942.88],[1.56807E-5,0.183625,-0.183619,0.965695],[-1,-3,0,0],[9E+09,9E+09,9E+09,9E+09,9E+09,9E+09]];
    CONST robtarget rB_t444 := [[-1995.85,-1995.91,1900.43],[0.689381,0.222581,-6.85382E-6,-0.689356],[-2,-2,-2,0],[9E+09,9E+09,9E+09,9E+09,9E+09,9E+09]];
    CONST robtarget rB_t444_c4 := [[-1995.85,-1995.91,1900.43],[0.689381,0.222581,-6.85382E-6,-0.689356],[0,-4,0,0],[9E+09,9E+09,9E+09,9E+09,9E+09,9E+09]];
    CONST robtarget rB_t444_c7 := [[-1995.85,-1995.91,1900.43],[0.689381,0.222581,-6.85382E-6,-0.689356],[0,-4,4,0],[9E+09,9E+09,9E+09,9E+09,9E+09,9E+09]];
    CONST jointtarget jA_t444 := [[-45.0007,0.818501,-33.7202,-180.001,26.9961,44.9993],[9E+09,9E+09,9E+09,9E+09,9E+09,9E+09]];
    CONST jointtarget jB_t444 := [[-134.999,57.5463,-68.0581,-179.999,53.7669,-134.999],[9E+09,9E+09,9E+09,9E+09,9E+09,9E+09]];
    CONST jointtarget jBseed_t444 := [[-134.999,57.5463,-68.0581,-179.999,53.7669,-134.999],[9E+09,9E+09,9E+09,9E+09,9E+09,9E+09]];

    CONST robtarget rA_t446 := [[1576.99,1577,183.348],[0.0233754,0.922155,0.381967,-0.0564366],[0,0,-2,0],[9E+09,9E+09,9E+09,9E+09,9E+09,9E+09]];
    CONST robtarget rB_t446 := [[1606.53,1606.49,1651.54],[0.550853,-6.74044E-6,0.627013,0.550832],[0,1,2,0],[9E+09,9E+09,9E+09,9E+09,9E+09,9E+09]];
    CONST robtarget rB_t446_c1 := [[1606.53,1606.49,1651.54],[0.550853,-6.74044E-6,0.627013,0.550832],[0,-4,-4,0],[9E+09,9E+09,9E+09,9E+09,9E+09,9E+09]];
    CONST robtarget rB_t446_c2 := [[1606.53,1606.49,1651.54],[0.550853,-6.74044E-6,0.627013,0.550832],[0,0,-4,0],[9E+09,9E+09,9E+09,9E+09,9E+09,9E+09]];
    CONST jointtarget jA_t446 := [[45.0003,46.6256,5.05326,0.00027126,45.3255,-180],[9E+09,9E+09,9E+09,9E+09,9E+09,9E+09]];
    CONST jointtarget jB_t446 := [[44.9992,12.1421,0.704976,179.999,25.1869,224.999],[9E+09,9E+09,9E+09,9E+09,9E+09,9E+09]];
    CONST jointtarget jBseed_t446 := [[44.9992,12.1421,0.704979,179.999,25.1869,224.999],[9E+09,9E+09,9E+09,9E+09,9E+09,9E+09]];

    CONST robtarget rA_t448 := [[83.3565,-460.282,2963.61],[0.0841153,-0.24427,0.314564,-0.913404],[-2,0,-3,0],[9E+09,9E+09,9E+09,9E+09,9E+09,9E+09]];
    CONST robtarget rB_t448 := [[-1614.19,-1614.21,520.711],[0.0272981,0.38171,0.921526,0.0659001],[-2,0,-1,0],[9E+09,9E+09,9E+09,9E+09,9E+09,9E+09]];
    CONST robtarget rB_t448_c5 := [[-1614.19,-1614.21,520.711],[0.0272981,0.38171,0.921526,0.0659001],[0,0,0,0],[9E+09,9E+09,9E+09,9E+09,9E+09,9E+09]];
    CONST jointtarget jA_t448 := [[-90.0003,-41.634,-10.3601,89.9997,29.9442,-180],[9E+09,9E+09,9E+09,9E+09,9E+09,9E+09]];
    CONST jointtarget jB_t448 := [[-135,37.9754,3.137,0.000226307,57.0684,-89.9998],[9E+09,9E+09,9E+09,9E+09,9E+09,9E+09]];
    CONST jointtarget jBseed_t448 := [[-135,37.9754,3.13699,0.000225867,57.0684,-89.9998],[9E+09,9E+09,9E+09,9E+09,9E+09,9E+09]];

    CONST robtarget rA_t449 := [[-1614.19,-1614.21,520.711],[0.0272981,0.38171,0.921526,0.0659001],[-2,0,-1,0],[9E+09,9E+09,9E+09,9E+09,9E+09,9E+09]];
    CONST robtarget rB_t449 := [[-15.7268,-1556.14,1431.23],[0.57729,0.719124,0.267024,-0.279812],[-2,-2,1,0],[9E+09,9E+09,9E+09,9E+09,9E+09,9E+09]];
    CONST robtarget rB_t449_c1 := [[-15.7268,-1556.14,1431.23],[0.57729,0.719124,0.267024,-0.279812],[0,-4,-4,0],[9E+09,9E+09,9E+09,9E+09,9E+09,9E+09]];
    CONST robtarget rB_t449_c2 := [[-15.7268,-1556.14,1431.23],[0.57729,0.719124,0.267024,-0.279812],[0,0,-4,0],[9E+09,9E+09,9E+09,9E+09,9E+09,9E+09]];
    CONST jointtarget jA_t449 := [[-135,37.9754,3.137,0.000226307,57.0684,-89.9998],[9E+09,9E+09,9E+09,9E+09,9E+09,9E+09]];
    CONST jointtarget jB_t449 := [[-90.0002,-24.8976,40.5576,-135,7.65038,180],[9E+09,9E+09,9E+09,9E+09,9E+09,9E+09]];
    CONST jointtarget jBseed_t449 := [[-90.0002,-24.8976,40.5576,-135,7.65038,180],[9E+09,9E+09,9E+09,9E+09,9E+09,9E+09]];

    CONST robtarget rA_t450 := [[-15.7268,-1556.14,1431.23],[0.57729,0.719124,0.267024,-0.279812],[-2,-2,1,0],[9E+09,9E+09,9E+09,9E+09,9E+09,9E+09]];
    CONST robtarget rB_t450 := [[1394.49,86.677,1479.93],[0.223577,-0.549711,-0.173763,-0.785899],[0,-3,-4,0],[9E+09,9E+09,9E+09,9E+09,9E+09,9E+09]];
    CONST robtarget rB_t450_c4 := [[1394.49,86.677,1479.93],[0.223577,-0.549711,-0.173763,-0.785899],[0,-4,0,0],[9E+09,9E+09,9E+09,9E+09,9E+09,9E+09]];
    CONST robtarget rB_t450_c5 := [[1394.49,86.677,1479.93],[0.223577,-0.549711,-0.173763,-0.785899],[0,0,0,0],[9E+09,9E+09,9E+09,9E+09,9E+09,9E+09]];
    CONST jointtarget jA_t450 := [[-90.0002,-24.8976,40.5576,-135,7.65038,180],[9E+09,9E+09,9E+09,9E+09,9E+09,9E+09]];
    CONST jointtarget jB_t450 := [[0.000746902,-32.7458,47.0324,-224.999,47.2115,-314.999],[9E+09,9E+09,9E+09,9E+09,9E+09,9E+09]];
    CONST jointtarget jBseed_t450 := [[0.000747185,-32.7458,47.0324,-224.999,47.2115,-314.999],[9E+09,9E+09,9E+09,9E+09,9E+09,9E+09]];

    CONST robtarget rA_t451 := [[1394.49,86.677,1479.93],[0.223577,-0.549711,-0.173763,-0.785899],[0,-3,-4,0],[9E+09,9E+09,9E+09,9E+09,9E+09,9E+09]];
    CONST robtarget rB_t451 := [[1524.7,-1381.29,1221.15],[0.796672,0.0602203,0.601398,-0.00273357],[-1,1,-2,0],[9E+09,9E+09,9E+09,9E+09,9E+09,9E+09]];
    CONST robtarget rB_t451_c4 := [[1524.7,-1381.29,1221.15],[0.796672,0.0602203,0.601398,-0.00273357],[0,-4,0,0],[9E+09,9E+09,9E+09,9E+09,9E+09,9E+09]];
    CONST jointtarget jA_t451 := [[0.000746902,-32.7458,47.0324,-224.999,47.2115,-314.999],[9E+09,9E+09,9E+09,9E+09,9E+09,9E+09]];
    CONST jointtarget jB_t451 := [[-44.9996,8.72891,21.2839,135,59.1668,-135],[9E+09,9E+09,9E+09,9E+09,9E+09,9E+09]];
    CONST jointtarget jBseed_t451 := [[-44.9996,8.7289,21.2839,135,59.1668,-135],[9E+09,9E+09,9E+09,9E+09,9E+09,9E+09]];

    CONST robtarget rA_t452 := [[1524.7,-1381.29,1221.15],[0.796672,0.0602203,0.601398,-0.00273357],[-1,1,-2,0],[9E+09,9E+09,9E+09,9E+09,9E+09,9E+09]];
    CONST robtarget rB_t452 := [[-0.0107167,-2875.01,1636.9],[0.629313,0.322429,0.322432,-0.629319],[-2,1,-3,0],[9E+09,9E+09,9E+09,9E+09,9E+09,9E+09]];
    CONST robtarget rB_t452_c2 := [[-0.0107167,-2875.01,1636.9],[0.629313,0.322429,0.322432,-0.629319],[0,0,-4,0],[9E+09,9E+09,9E+09,9E+09,9E+09,9E+09]];
    CONST jointtarget jA_t452 := [[-44.9996,8.72891,21.2839,135,59.1668,-135],[9E+09,9E+09,9E+09,9E+09,9E+09,9E+09]];
    CONST jointtarget jB_t452 := [[-90.0002,50.7565,-49.3081,180,37.1917,-180],[9E+09,9E+09,9E+09,9E+09,9E+09,9E+09]];
    CONST jointtarget jBseed_t452 := [[-90.0002,50.7566,-49.3081,180,37.1917,-180],[9E+09,9E+09,9E+09,9E+09,9E+09,9E+09]];

    CONST robtarget rA_t455 := [[0.00233704,1928.96,133.762],[0.0199452,0.382164,-0.922624,0.0481527],[0,-1,0,0],[9E+09,9E+09,9E+09,9E+09,9E+09,9E+09]];
    CONST robtarget rB_t455 := [[-1944.95,1890.68,1605.67],[0.65049,-0.20912,-0.708424,-0.176824],[1,-4,-4,0],[9E+09,9E+09,9E+09,9E+09,9E+09,9E+09]];
    CONST robtarget rB_t455_c4 := [[-1944.95,1890.68,1605.67],[0.65049,-0.20912,-0.708424,-0.176824],[0,-4,0,0],[9E+09,9E+09,9E+09,9E+09,9E+09,9E+09]];
    CONST robtarget rB_t455_c5 := [[-1944.95,1890.68,1605.67],[0.65049,-0.20912,-0.708424,-0.176824],[0,0,0,0],[9E+09,9E+09,9E+09,9E+09,9E+09,9E+09]];
    CONST jointtarget jA_t455 := [[89.9999,38.2061,22.4067,-7.23746E-5,35.3624,44.9999],[9E+09,9E+09,9E+09,9E+09,9E+09,9E+09]];
    CONST jointtarget jB_t455 := [[135,36.8035,-31.427,-270,13.2902,-270],[9E+09,9E+09,9E+09,9E+09,9E+09,9E+09]];
    CONST jointtarget jBseed_t455 := [[135,36.8035,-31.427,-270,13.2902,-270],[9E+09,9E+09,9E+09,9E+09,9E+09,9E+09]];

    CONST robtarget rA_t461 := [[-1042,-1042.01,2491.64],[0.356122,0.338249,0.140104,-0.85973],[-2,-2,2,0],[9E+09,9E+09,9E+09,9E+09,9E+09,9E+09]];
    CONST robtarget rB_t461 := [[126.577,-1680.89,357.926],[0.0520461,0.853162,-0.242274,0.459031],[-2,0,-4,0],[9E+09,9E+09,9E+09,9E+09,9E+09,9E+09]];
    CONST robtarget rB_t461_c4 := [[126.577,-1680.89,357.926],[0.0520461,0.853162,-0.242274,0.459031],[0,-4,0,0],[9E+09,9E+09,9E+09,9E+09,9E+09,9E+09]];
    CONST robtarget rB_t461_c5 := [[126.577,-1680.89,357.926],[0.0520461,0.853162,-0.242274,0.459031],[0,0,0,0],[9E+09,9E+09,9E+09,9E+09,9E+09,9E+09]];
    CONST jointtarget jA_t461 := [[-135,-19.8621,2.76803,-180,29.9533,180],[9E+09,9E+09,9E+09,9E+09,9E+09,9E+09]];
    CONST jointtarget jB_t461 := [[-90.0005,20.6348,40.8631,89.9995,49.2917,-315.001],[9E+09,9E+09,9E+09,9E+09,9E+09,9E+09]];
    CONST jointtarget jBseed_t461 := [[-90.0005,20.6348,40.8631,89.9995,49.2917,-315.001],[9E+09,9E+09,9E+09,9E+09,9E+09,9E+09]];

    CONST robtarget rA_t462 := [[126.577,-1680.89,357.926],[0.0520461,0.853162,-0.242274,0.459031],[-2,0,-4,0],[9E+09,9E+09,9E+09,9E+09,9E+09,9E+09]];
    CONST robtarget rB_t462 := [[2177.52,136.908,1496.14],[0.637379,-0.697821,0.306198,-0.11418],[0,1,-2,0],[9E+09,9E+09,9E+09,9E+09,9E+09,9E+09]];
    CONST robtarget rB_t462_c2 := [[2177.52,136.908,1496.14],[0.637379,-0.697821,0.306198,-0.11418],[0,0,-4,0],[9E+09,9E+09,9E+09,9E+09,9E+09,9E+09]];
    CONST jointtarget jA_t462 := [[-90.0005,20.6348,40.8631,89.9995,49.2917,-315.001],[9E+09,9E+09,9E+09,9E+09,9E+09,9E+09]];
    CONST jointtarget jB_t462 := [[0.000814675,11.5671,4.79935,90.0008,55.0468,-179.999],[9E+09,9E+09,9E+09,9E+09,9E+09,9E+09]];
    CONST jointtarget jBseed_t462 := [[0.000814447,11.5671,4.79934,90.0008,55.0468,-179.999],[9E+09,9E+09,9E+09,9E+09,9E+09,9E+09]];

    CONST robtarget rA_t463 := [[2177.52,136.908,1496.14],[0.637379,-0.697821,0.306198,-0.11418],[0,1,-2,0],[9E+09,9E+09,9E+09,9E+09,9E+09,9E+09]];
    CONST robtarget rB_t463 := [[1406.9,1507.89,-175.697],[0.440792,-0.841613,0.306654,0.0579034],[0,-3,-3,0],[9E+09,9E+09,9E+09,9E+09,9E+09,9E+09]];
    CONST robtarget rB_t463_c2 := [[1406.9,1507.89,-175.697],[0.440792,-0.841613,0.306654,0.0579034],[0,0,-4,0],[9E+09,9E+09,9E+09,9E+09,9E+09,9E+09]];
    CONST jointtarget jA_t463 := [[0.000814675,11.5671,4.79935,90.0008,55.0468,-179.999],[9E+09,9E+09,9E+09,9E+09,9E+09,9E+09]];
    CONST jointtarget jB_t463 := [[45.0006,54.9242,15.2812,-224.999,37.199,-224.999],[9E+09,9E+09,9E+09,9E+09,9E+09,9E+09]];
    CONST jointtarget jBseed_t463 := [[45.0006,54.9242,15.2812,-224.999,37.199,-224.999],[9E+09,9E+09,9E+09,9E+09,9E+09,9E+09]];

    CONST robtarget rA_t465 := [[1566.54,1425.49,2737.66],[0.355531,-0.68129,0.308403,-0.560651],[0,-1,2,0],[9E+09,9E+09,9E+09,9E+09,9E+09,9E+09]];
    CONST robtarget rB_t465 := [[574.565,-627.773,2106.19],[0.743062,0.29642,0.468192,-0.37522],[-1,-2,-4,0],[9E+09,9E+09,9E+09,9E+09,9E+09,9E+09]];
    CONST robtarget rB_t465_c5 := [[574.565,-627.773,2106.19],[0.743062,0.29642,0.468192,-0.37522],[0,0,0,0],[9E+09,9E+09,9E+09,9E+09,9E+09,9E+09]];
    CONST jointtarget jA_t465 := [[45,32.3209,-71.9462,-45,57.6287,270],[9E+09,9E+09,9E+09,9E+09,9E+09,9E+09]];
    CONST jointtarget jB_t465 := [[-45.0008,-59.0954,35.7649,-90.0008,13.0155,-270.001],[9E+09,9E+09,9E+09,9E+09,9E+09,9E+09]];
    CONST jointtarget jBseed_t465 := [[-45.0008,-59.0954,35.7649,-90.0008,13.0155,-270.001],[9E+09,9E+09,9E+09,9E+09,9E+09,9E+09]];

    CONST robtarget rA_t467 := [[1287.38,1138.58,-3.37622],[0.330421,0.694365,0.623434,0.141454],[0,2,2,0],[9E+09,9E+09,9E+09,9E+09,9E+09,9E+09]];
    CONST robtarget rB_t467 := [[1645.77,1585.99,1729.58],[0.0980131,0.529509,0.411551,0.735282],[0,-2,-2,0],[9E+09,9E+09,9E+09,9E+09,9E+09,9E+09]];
    CONST robtarget rB_t467_c8 := [[1645.77,1585.99,1729.58],[0.0980131,0.529509,0.411551,0.735282],[0,0,4,0],[9E+09,9E+09,9E+09,9E+09,9E+09,9E+09]];
    CONST jointtarget jA_t467 := [[44.9995,39.1217,33.6146,270,39.0484,225],[9E+09,9E+09,9E+09,9E+09,9E+09,9E+09]];
    CONST jointtarget jB_t467 := [[45,12.6328,-3.42905,-135,20.9735,-90],[9E+09,9E+09,9E+09,9E+09,9E+09,9E+09]];
    CONST jointtarget jBseed_t467 := [[45,12.6328,-3.42905,-135,20.9735,-90],[9E+09,9E+09,9E+09,9E+09,9E+09,9E+09]];

    CONST robtarget rA_t468 := [[1645.77,1585.99,1729.58],[0.0980131,0.529509,0.411551,0.735282],[0,-2,-2,0],[9E+09,9E+09,9E+09,9E+09,9E+09,9E+09]];
    CONST robtarget rB_t468 := [[2229.59,-0.00201698,2773.73],[0.659696,0.254562,0.254562,0.659695],[-1,1,2,0],[9E+09,9E+09,9E+09,9E+09,9E+09,9E+09]];
    CONST robtarget rB_t468_c4 := [[2229.59,-0.00201698,2773.73],[0.659696,0.254562,0.254562,0.659695],[0,-4,0,0],[9E+09,9E+09,9E+09,9E+09,9E+09,9E+09]];
    CONST robtarget rB_t468_c7 := [[2229.59,-0.00201698,2773.73],[0.659696,0.254562,0.254562,0.659695],[0,-4,4,0],[9E+09,9E+09,9E+09,9E+09,9E+09,9E+09]];
    CONST jointtarget jA_t468 := [[45,12.6328,-3.42905,-135,20.9735,-90],[9E+09,9E+09,9E+09,9E+09,9E+09,9E+09]];
    CONST jointtarget jB_t468 := [[-5.2556E-5,37.6275,-74.7273,180,10.6992,270],[9E+09,9E+09,9E+09,9E+09,9E+09,9E+09]];
    CONST jointtarget jBseed_t468 := [[-5.25223E-5,37.6275,-74.7273,180,10.6992,270],[9E+09,9E+09,9E+09,9E+09,9E+09,9E+09]];

    CONST robtarget rA_t469 := [[2229.59,-0.00201698,2773.73],[0.659696,0.254562,0.254562,0.659695],[-1,1,2,0],[9E+09,9E+09,9E+09,9E+09,9E+09,9E+09]];
    CONST robtarget rB_t469 := [[-82.0683,-1902.26,1972.08],[0.609307,0.358823,-0.611887,0.354381],[-2,-2,-2,0],[9E+09,9E+09,9E+09,9E+09,9E+09,9E+09]];
    CONST robtarget rB_t469_c9 := [[-82.0683,-1902.26,1972.08],[0.609307,0.358823,-0.611887,0.354381],[0,4,4,0],[9E+09,9E+09,9E+09,9E+09,9E+09,9E+09]];
    CONST jointtarget jA_t469 := [[-5.2556E-5,37.6275,-74.7273,180,10.6992,270],[9E+09,9E+09,9E+09,9E+09,9E+09,9E+09]];
    CONST jointtarget jB_t469 := [[-90.0005,-5.74419,6.16015,-90.0005,29.4278,-90.0005],[9E+09,9E+09,9E+09,9E+09,9E+09,9E+09]];
    CONST jointtarget jBseed_t469 := [[-90.0005,-5.74419,6.16016,-90.0005,29.4278,-90.0005],[9E+09,9E+09,9E+09,9E+09,9E+09,9E+09]];

    CONST robtarget rA_t470 := [[-82.0683,-1902.26,1972.08],[0.609307,0.358823,-0.611887,0.354381],[-2,-2,-2,0],[9E+09,9E+09,9E+09,9E+09,9E+09,9E+09]];
    CONST robtarget rB_t470 := [[-0.00742192,-1363.62,2049.39],[6.35341E-6,2.03801E-6,-0.543879,0.839164],[-2,-3,-4,0],[9E+09,9E+09,9E+09,9E+09,9E+09,9E+09]];
    CONST robtarget rB_t470_c1 := [[-0.00742192,-1363.62,2049.39],[6.35341E-6,2.03801E-6,-0.543879,0.839164],[0,-4,-4,0],[9E+09,9E+09,9E+09,9E+09,9E+09,9E+09]];
    CONST robtarget rB_t470_c4 := [[-0.00742192,-1363.62,2049.39],[6.35341E-6,2.03801E-6,-0.543879,0.839164],[0,-4,0,0],[9E+09,9E+09,9E+09,9E+09,9E+09,9E+09]];
    CONST jointtarget jA_t470 := [[-90.0005,-5.74419,6.16015,-90.0005,29.4278,-90.0005],[9E+09,9E+09,9E+09,9E+09,9E+09,9E+09]];
    CONST jointtarget jB_t470 := [[-90.0003,-33.7492,27.0208,-180,17.3754,-270],[9E+09,9E+09,9E+09,9E+09,9E+09,9E+09]];
    CONST jointtarget jBseed_t470 := [[-90.0003,-33.7492,27.0208,-180,17.3754,-270],[9E+09,9E+09,9E+09,9E+09,9E+09,9E+09]];

    CONST robtarget rA_t472 := [[1670.37,1553.97,70.707],[0.24436,0.706763,0.603939,0.27574],[0,-1,-2,0],[9E+09,9E+09,9E+09,9E+09,9E+09,9E+09]];
    CONST robtarget rB_t472 := [[1698.07,121.103,3070.64],[0.501556,-0.0205597,0.498446,0.706802],[-1,-4,3,0],[9E+09,9E+09,9E+09,9E+09,9E+09,9E+09]];
    CONST robtarget rB_t472_c4 := [[1698.07,121.103,3070.64],[0.501556,-0.0205597,0.498446,0.706802],[0,-4,0,0],[9E+09,9E+09,9E+09,9E+09,9E+09,9E+09]];
    CONST robtarget rB_t472_c5 := [[1698.07,121.103,3070.64],[0.501556,-0.0205597,0.498446,0.706802],[0,0,0,0],[9E+09,9E+09,9E+09,9E+09,9E+09,9E+09]];
    CONST jointtarget jA_t472 := [[45.0007,50.7346,6.12842,-89.9993,29.5413,-134.999],[9E+09,9E+09,9E+09,9E+09,9E+09,9E+09]];
    CONST jointtarget jB_t472 := [[-0.000364208,20.2063,-67.0504,-270,46.4882,360],[9E+09,9E+09,9E+09,9E+09,9E+09,9E+09]];
    CONST jointtarget jBseed_t472 := [[-0.0003643,20.2063,-67.0504,-270,46.4882,360],[9E+09,9E+09,9E+09,9E+09,9E+09,9E+09]];

    CONST robtarget rA_t473 := [[1698.07,121.103,3070.64],[0.501556,-0.0205597,0.498446,0.706802],[-1,-4,3,0],[9E+09,9E+09,9E+09,9E+09,9E+09,9E+09]];
    CONST robtarget rB_t473 := [[-1766.92,1736.68,2488.45],[0.801534,-0.411131,-0.229574,0.368525],[1,-3,1,0],[9E+09,9E+09,9E+09,9E+09,9E+09,9E+09]];
    CONST robtarget rB_t473_c4 := [[-1766.92,1736.68,2488.45],[0.801534,-0.411131,-0.229574,0.368525],[0,-4,0,0],[9E+09,9E+09,9E+09,9E+09,9E+09,9E+09]];
    CONST jointtarget jA_t473 := [[-0.000364208,20.2063,-67.0504,-270,46.4882,360],[9E+09,9E+09,9E+09,9E+09,9E+09,9E+09]];
    CONST jointtarget jB_t473 := [[135,40.5353,-67.2488,-225,10.4392,135],[9E+09,9E+09,9E+09,9E+09,9E+09,9E+09]];
    CONST jointtarget jBseed_t473 := [[135,40.5353,-67.2488,-225,10.4392,135],[9E+09,9E+09,9E+09,9E+09,9E+09,9E+09]];

    CONST robtarget rA_t474 := [[-1766.92,1736.68,2488.45],[0.801534,-0.411131,-0.229574,0.368525],[1,-3,1,0],[9E+09,9E+09,9E+09,9E+09,9E+09,9E+09]];
    CONST robtarget rB_t474 := [[-135.791,1608.72,1301.46],[0.601781,-0.586193,-0.5176,0.16226],[0,-4,-3,0],[9E+09,9E+09,9E+09,9E+09,9E+09,9E+09]];
    CONST robtarget rB_t474_c4 := [[-135.791,1608.72,1301.46],[0.601781,-0.586193,-0.5176,0.16226],[0,-4,0,0],[9E+09,9E+09,9E+09,9E+09,9E+09,9E+09]];
    CONST robtarget rB_t474_c5 := [[-135.791,1608.72,1301.46],[0.601781,-0.586193,-0.5176,0.16226],[0,0,0,0],[9E+09,9E+09,9E+09,9E+09,9E+09,9E+09]];
    CONST jointtarget jA_t474 := [[135,40.5353,-67.2488,-225,10.4392,135],[9E+09,9E+09,9E+09,9E+09,9E+09,9E+09]];
    CONST jointtarget jB_t474 := [[89.9995,-15.9105,38.4469,-270,54.4096,-225],[9E+09,9E+09,9E+09,9E+09,9E+09,9E+09]];
    CONST jointtarget jBseed_t474 := [[89.9995,-15.9105,38.4469,-270,54.4096,-225],[9E+09,9E+09,9E+09,9E+09,9E+09,9E+09]];

    CONST robtarget rA_t475 := [[-135.791,1608.72,1301.46],[0.601781,-0.586193,-0.5176,0.16226],[0,-4,-3,0],[9E+09,9E+09,9E+09,9E+09,9E+09,9E+09]];
    CONST robtarget rB_t475 := [[1798.02,1723.9,531.198],[0.238469,0.42684,0.850128,0.195507],[0,-1,-3,0],[9E+09,9E+09,9E+09,9E+09,9E+09,9E+09]];
    CONST robtarget rB_t475_c2 := [[1798.02,1723.9,531.198],[0.238469,0.42684,0.850128,0.195507],[0,0,-4,0],[9E+09,9E+09,9E+09,9E+09,9E+09,9E+09]];
    CONST jointtarget jA_t475 := [[89.9995,-15.9105,38.4469,-270,54.4096,-225],[9E+09,9E+09,9E+09,9E+09,9E+09,9E+09]];
    CONST jointtarget jB_t475 := [[44.9991,42.9048,-3.6671,-45.0009,26.3277,-225.001],[9E+09,9E+09,9E+09,9E+09,9E+09,9E+09]];
    CONST jointtarget jBseed_t475 := [[44.9991,42.9048,-3.6671,-45.0009,26.3277,-225.001],[9E+09,9E+09,9E+09,9E+09,9E+09,9E+09]];

    CONST robtarget rA_t477 := [[-0.0223292,-2304.88,1581.76],[0.526261,0.759348,-0.314528,0.217975],[-2,-1,-3,0],[9E+09,9E+09,9E+09,9E+09,9E+09,9E+09]];
    CONST robtarget rB_t477 := [[-69.6204,-1624.2,1584.64],[0.659331,0.336651,-0.528318,0.415728],[-2,2,3,0],[9E+09,9E+09,9E+09,9E+09,9E+09,9E+09]];
    CONST robtarget rB_t477_c4 := [[-69.6204,-1624.2,1584.64],[0.659331,0.336651,-0.528318,0.415728],[0,-4,0,0],[9E+09,9E+09,9E+09,9E+09,9E+09,9E+09]];
    CONST jointtarget jA_t477 := [[-90.0005,14.0794,-2.45308,-0.000547372,8.92666,-225.001],[9E+09,9E+09,9E+09,9E+09,9E+09,9E+09]];
    CONST jointtarget jB_t477 := [[-90.0008,-20.6201,34.2216,224.999,36.1132,314.999],[9E+09,9E+09,9E+09,9E+09,9E+09,9E+09]];
    CONST jointtarget jBseed_t477 := [[-90.0008,-20.6201,34.2216,224.999,36.1132,314.999],[9E+09,9E+09,9E+09,9E+09,9E+09,9E+09]];

    CONST robtarget rA_t479 := [[251.84,103.584,2724.4],[0.707096,0.31481,0.306087,0.554275],[0,-2,1,0],[9E+09,9E+09,9E+09,9E+09,9E+09,9E+09]];
    CONST robtarget rB_t479 := [[-98.1109,903.889,3290.74],[0.266575,-0.377919,0.139435,0.875599],[1,1,3,0],[9E+09,9E+09,9E+09,9E+09,9E+09,9E+09]];
    CONST robtarget rB_t479_c7 := [[-98.1109,903.889,3290.74],[0.266575,-0.377919,0.139435,0.875599],[0,-4,4,0],[9E+09,9E+09,9E+09,9E+09,9E+09,9E+09]];
    CONST jointtarget jA_t479 := [[44.999,-57.1471,5.02946,-90.001,38.8818,134.999],[9E+09,9E+09,9E+09,9E+09,9E+09,9E+09]];
    CONST jointtarget jB_t479 := [[90.0002,-9.03287,-47.5506,90.0002,35.9777,315],[9E+09,9E+09,9E+09,9E+09,9E+09,9E+09]];
    CONST jointtarget jBseed_t479 := [[90.0002,-9.03287,-47.5506,90.0002,35.9777,315],[9E+09,9E+09,9E+09,9E+09,9E+09,9E+09]];

    CONST robtarget rA_t481 := [[1795.92,-1913.67,587.316],[0.0955417,0.478729,0.820833,-0.29652],[-1,-1,-4,0],[9E+09,9E+09,9E+09,9E+09,9E+09,9E+09]];
    CONST robtarget rB_t481 := [[-652.406,-631.961,3432.88],[0.367965,0.17558,0.0268566,-0.912717],[-2,-2,-3,0],[9E+09,9E+09,9E+09,9E+09,9E+09,9E+09]];
    CONST robtarget rB_t481_c2 := [[-652.406,-631.961,3432.88],[0.367965,0.17558,0.0268566,-0.912717],[0,0,-4,0],[9E+09,9E+09,9E+09,9E+09,9E+09,9E+09]];
    CONST jointtarget jA_t481 := [[-44.9993,49.0756,-15.8034,-44.9993,44.8567,-314.999],[9E+09,9E+09,9E+09,9E+09,9E+09,9E+09]];
    CONST jointtarget jB_t481 := [[-134.999,3.19528,-68.3318,-134.999,7.03696,-224.999],[9E+09,9E+09,9E+09,9E+09,9E+09,9E+09]];
    CONST jointtarget jBseed_t481 := [[-134.999,3.19529,-68.3319,-134.999,7.03696,-224.999],[9E+09,9E+09,9E+09,9E+09,9E+09,9E+09]];

    CONST robtarget rA_t482 := [[-652.406,-631.961,3432.88],[0.367965,0.17558,0.0268566,-0.912717],[-2,-2,-3,0],[9E+09,9E+09,9E+09,9E+09,9E+09,9E+09]];
    CONST robtarget rB_t482 := [[24.2868,-992.068,2739.09],[0.0334906,-0.0649989,0.520641,-0.850639],[-2,0,2,0],[9E+09,9E+09,9E+09,9E+09,9E+09,9E+09]];
    CONST robtarget rB_t482_c2 := [[24.2868,-992.068,2739.09],[0.0334906,-0.0649989,0.520641,-0.850639],[0,0,-4,0],[9E+09,9E+09,9E+09,9E+09,9E+09,9E+09]];
    CONST jointtarget jA_t482 := [[-134.999,3.19528,-68.3318,-134.999,7.03696,-224.999],[9E+09,9E+09,9E+09,9E+09,9E+09,9E+09]];
    CONST jointtarget jB_t482 := [[-90.0003,-33.5734,-1.89763,44.9997,11.8711,225],[9E+09,9E+09,9E+09,9E+09,9E+09,9E+09]];
    CONST jointtarget jBseed_t482 := [[-90.0003,-33.5734,-1.89764,44.9997,11.8711,225],[9E+09,9E+09,9E+09,9E+09,9E+09,9E+09]];

    CONST robtarget rA_t483 := [[24.2868,-992.068,2739.09],[0.0334906,-0.0649989,0.520641,-0.850639],[-2,0,2,0],[9E+09,9E+09,9E+09,9E+09,9E+09,9E+09]];
    CONST robtarget rB_t483 := [[733.459,733.478,2508.95],[0.85326,-0.354275,0.146751,-0.353412],[0,-2,1,0],[9E+09,9E+09,9E+09,9E+09,9E+09,9E+09]];
    CONST robtarget rB_t483_c4 := [[733.459,733.478,2508.95],[0.85326,-0.354275,0.146751,-0.353412],[0,-4,0,0],[9E+09,9E+09,9E+09,9E+09,9E+09,9E+09]];
    CONST jointtarget jA_t483 := [[-90.0003,-33.5734,-1.89763,44.9997,11.8711,225],[9E+09,9E+09,9E+09,9E+09,9E+09,9E+09]];
    CONST jointtarget jB_t483 := [[45.0008,-39.1839,13.4126,-179.999,19.1314,90.0008],[9E+09,9E+09,9E+09,9E+09,9E+09,9E+09]];
    CONST jointtarget jBseed_t483 := [[45.0008,-39.1839,13.4126,-179.999,19.1314,90.0008],[9E+09,9E+09,9E+09,9E+09,9E+09,9E+09]];

    CONST robtarget rA_t484 := [[733.459,733.478,2508.95],[0.85326,-0.354275,0.146751,-0.353412],[0,-2,1,0],[9E+09,9E+09,9E+09,9E+09,9E+09,9E+09]];
    CONST robtarget rB_t484 := [[864.724,864.744,3072.98],[0.363593,-0.288274,-0.119404,-0.877748],[0,2,0,0],[9E+09,9E+09,9E+09,9E+09,9E+09,9E+09]];
    CONST robtarget rB_t484_c4 := [[864.724,864.744,3072.98],[0.363593,-0.288274,-0.119404,-0.877748],[0,-4,0,0],[9E+09,9E+09,9E+09,9E+09,9E+09,9E+09]];
    CONST robtarget rB_t484_c7 := [[864.724,864.744,3072.98],[0.363593,-0.288274,-0.119404,-0.877748],[0,-4,4,0],[9E+09,9E+09,9E+09,9E+09,9E+09,9E+09]];
    CONST jointtarget jA_t484 := [[45.0008,-39.1839,13.4126,-179.999,19.1314,90.0008],[9E+09,9E+09,9E+09,9E+09,9E+09,9E+09]];
    CONST jointtarget jB_t484 := [[45.0007,-11.6733,-29.6298,180.001,12.3344,0.000680984],[9E+09,9E+09,9E+09,9E+09,9E+09,9E+09]];
    CONST jointtarget jBseed_t484 := [[45.0007,-11.6733,-29.6298,180.001,12.3344,0.000684011],[9E+09,9E+09,9E+09,9E+09,9E+09,9E+09]];

    CONST robtarget rA_t485 := [[864.724,864.744,3072.98],[0.363593,-0.288274,-0.119404,-0.877748],[0,2,0,0],[9E+09,9E+09,9E+09,9E+09,9E+09,9E+09]];
    CONST robtarget rB_t485 := [[-156.188,32.3569,3418.1],[0.820893,-0.20476,-0.394721,0.358334],[1,0,2,0],[9E+09,9E+09,9E+09,9E+09,9E+09,9E+09]];
    CONST robtarget rB_t485_c2 := [[-156.188,32.3569,3418.1],[0.820893,-0.20476,-0.394721,0.358334],[0,0,-4,0],[9E+09,9E+09,9E+09,9E+09,9E+09,9E+09]];
    CONST robtarget rB_t485_c5 := [[-156.188,32.3569,3418.1],[0.820893,-0.20476,-0.394721,0.358334],[0,0,0,0],[9E+09,9E+09,9E+09,9E+09,9E+09,9E+09]];
    CONST jointtarget jA_t485 := [[45.0007,-11.6733,-29.6298,180.001,12.3344,0.000680984],[9E+09,9E+09,9E+09,9E+09,9E+09,9E+09]];
    CONST jointtarget jB_t485 := [[135,-13.9732,-69.2642,45,47.8597,225],[9E+09,9E+09,9E+09,9E+09,9E+09,9E+09]];
    CONST jointtarget jBseed_t485 := [[135,-13.9732,-69.2642,45,47.8597,225],[9E+09,9E+09,9E+09,9E+09,9E+09,9E+09]];

